KUKA KRL program: MyProgram_213().src

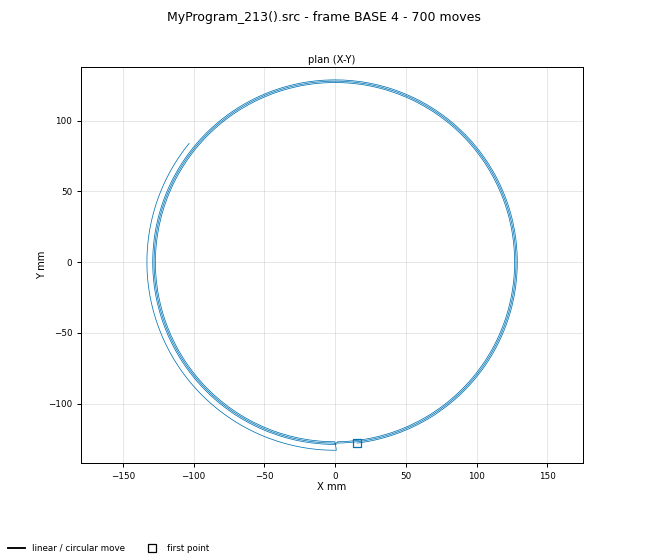
[picture p0: tool path of MyProgram_213().src in frame BASE 4, 700 of 700 moves have a stored position in this frame; points joined in program order, loops and branches not executed]
&ACCESS RVP
&REL 1
&PARAM TEMPLATE = C:\KRC\Roboter\Template\vorgabe
&PARAM EDITMASK = *
DEF MyProgram_213()
; ---- Setting reference (Base) ----
$BASE = BASE_DATA[4]

; --------------------------
; ---- Setting tool (TCP) ----
$TOOL = TOOL_DATA[3]
; --------------------------

$VEL.CP = VEL_APROX_PRINT
Startdeposition()
$VEL.CP = VEL_PRINT
LIN {X 15.6631,Y -127.8764,Z 150,A -84.7051,B 21.2641,C -0.7422,E1 21.2973,E2 532.2329} C_DIS
LIN {X 18.2596,Y -127.5309,Z 150,A -82.9319,B 21.2632,C -0.7696,E1 21.3024,E2 530.386} C_DIS
LIN {X 22.8874,Y -126.7822,Z 150,A -81.4703,B 21.2641,C -0.7437,E1 21.3063,E2 528.9976} C_DIS
LIN {X 26.4582,Y -126.0874,Z 150,A -79.8315,B 21.2641,C -0.746,E1 21.3107,E2 527.3551} C_DIS
LIN {X 29.8823,Y -125.3182,Z 150,A -78.1484,B 21.2638,C -0.7528,E1 21.3154,E2 525.6559} C_DIS
LIN {X 34.3471,Y -124.1689,Z 150,A -76.3006,B 21.264,C -0.746,E1 21.3203,E2 523.8305} C_DIS
LIN {X 37.1802,Y -123.3508,Z 150,A -74.8395,B 21.2637,C -0.754,E1 21.3243,E2 522.3503} C_DIS
LIN {X 39.8601,Y -122.5118,Z 150,A -73.2468,B 21.2632,C -0.7707,E1 21.3286,E2 520.7152} C_DIS
LIN {X 43.4,Y -121.3013,Z 150,A -71.878,B 21.2635,C -0.7597,E1 21.3321,E2 519.3802} C_DIS
LIN {X 46.1763,Y -120.2726,Z 150,A -69.6143,B 21.262,C -0.8039,E1 21.3384,E2 517.0006} C_DIS
LIN {X 52.7771,Y -117.5247,Z 150,A -67.5502,B 21.2636,C -0.7583,E1 21.3433,E2 515.068} C_DIS
LIN {X 56.4516,Y -115.806,Z 150,A -65.6853,B 21.2634,C -0.7638,E1 21.348,E2 513.1938} C_DIS
LIN {X 59.7288,Y -114.1488,Z 150,A -64.1905,B 21.2635,C -0.7603,E1 21.3516,E2 511.7136} C_DIS
LIN {X 62.0762,Y -112.8921,Z 150,A -62.4263,B 21.2625,C -0.7884,E1 21.3561,E2 509.8784} C_DIS
LIN {X 65.7163,Y -110.8119,Z 150,A -60.7738,B 21.2628,C -0.7822,E1 21.3601,E2 508.2491} C_DIS
LIN {X 68.4873,Y -109.1217,Z 150,A -59.507,B 21.2629,C -0.7768,E1 21.363,E2 507.0018} C_DIS
LIN {X 72.1434,Y -106.7393,Z 150,A -57.4433,B 21.2626,C -0.7862,E1 21.3678,E2 504.9208} C_DIS
LIN {X 79.2097,Y -101.6066,Z 150,A -52.9654,B 21.2614,C -0.8213,E1 21.378,E2 500.3657} C_DIS
LIN {X 83.9285,Y -97.7445,Z 150,A -51.3313,B 21.2629,C -0.7781,E1 21.3812,E2 498.8579} C_DIS
LIN {X 88.2018,Y -93.9067,Z 150,A -48.6114,B 21.2624,C -0.7913,E1 21.3869,E2 496.1147} C_DIS
LIN {X 93.8183,Y -88.2955,Z 150,A -45.2617,B 21.2624,C -0.7915,E1 21.3935,E2 492.7815} C_DIS
LIN {X 97.7896,Y -83.8762,Z 150,A -42.3753,B 21.2618,C -0.8092,E1 21.3989,E2 489.8621} C_DIS
LIN {X 100.2723,Y -80.8914,Z 150,A -39.8306,B 21.2602,C -0.8514,E1 21.4035,E2 487.2158} C_DIS
LIN {X 104.1395,Y -75.8485,Z 150,A -37.8772,B 21.2615,C -0.8186,E1 21.4066,E2 485.3636} C_DIS
LIN {X 106.3473,Y -72.7204,Z 150,A -36.1507,B 21.2612,C -0.8244,E1 21.4093,E2 483.6315} C_DIS
LIN {X 108.4584,Y -69.5322,Z 150,A -34.4696,B 21.2612,C -0.8282,E1 21.4119,E2 481.95} C_DIS
LIN {X 110.584,Y -66.0994,Z 150,A -32.5234,B 21.2607,C -0.8402,E1 21.4147,E2 479.9828} C_DIS
LIN {X 113.2426,Y -61.434,Z 150,A -30.2698,B 21.2607,C -0.8408,E1 21.4178,E2 477.7415} C_DIS
LIN {X 114.9781,Y -58.1173,Z 150,A -28.251,B 21.2598,C -0.8621,E1 21.4204,E2 475.6772} C_DIS
LIN {X 116.8181,Y -54.3235,Z 150,A -26.8866,B 21.2605,C -0.844,E1 21.4219,E2 474.3712} C_DIS
LIN {X 118.3125,Y -50.9865,Z 150,A -25.2141,B 21.2602,C -0.851,E1 21.4238,E2 472.6904} C_DIS
LIN {X 119.5881,Y -47.9188,Z 150,A -23.3605,B 21.2594,C -0.8729,E1 21.4258,E2 470.7892} C_DIS
LIN {X 121.0232,Y -44.1714,Z 150,A -21.9784,B 21.2599,C -0.8597,E1 21.4271,E2 469.4525} C_DIS
LIN {X 122.1969,Y -40.8095,Z 150,A -20.5058,B 21.2599,C -0.8594,E1 21.4284,E2 467.9905} C_DIS
LIN {X 123.1384,Y -37.8741,Z 150,A -18.6791,B 21.2589,C -0.8848,E1 21.4299,E2 466.1068} C_DIS
LIN {X 124.2425,Y -34.084,Z 150,A -17.3486,B 21.2595,C -0.8705,E1 21.4309,E2 464.8245} C_DIS
LIN {X 125.1127,Y -30.7349,Z 150,A -15.7365,B 21.2592,C -0.8787,E1 21.432,E2 463.2011} C_DIS
LIN {X 125.9433,Y -27.1259,Z 150,A -14.1941,B 21.2592,C -0.8791,E1 21.4329,E2 461.6684} C_DIS
LIN {X 126.4726,Y -24.5423,Z 150,A -12.9669,B 21.2589,C -0.8853,E1 21.4336,E2 460.4328} C_DIS
LIN {X 127.608,Y -17.7203,Z 150,A -10.3865,B 21.2594,C -0.8721,E1 21.4348,E2 457.9065} C_DIS
LIN {X 128.361,Y -11.0017,Z 150,A -7.2717,B 21.2589,C -0.8865,E1 21.4357,E2 454.7743} C_DIS
LIN {X 128.759,Y -4.3743,Z 150,A -4.1384,B 21.2581,C -0.9042,E1 21.4362,E2 451.615} C_DIS
LIN {X 128.8171,Y 1.9443,Z 150,A -0.5419,B 21.2563,C -0.9496,E1 21.4362,E2 447.9196} C_DIS
LIN {X 128.6186,Y 7.4224,Z 150,A 1.2036,B 21.2573,C -0.9251,E1 21.4359,E2 446.2535} C_DIS
LIN {X 127.9217,Y 15.2834,Z 150,A 4.5209,B 21.2572,C -0.9273,E1 21.4351,E2 442.9539} C_DIS
LIN {X 127.0644,Y 21.2642,Z 150,A 7.3154,B 21.2566,C -0.9405,E1 21.4339,E2 440.1427} C_DIS
LIN {X 125.7034,Y 28.2204,Z 150,A 10.2724,B 21.2566,C -0.9412,E1 21.4323,E2 437.2044} C_DIS
LIN {X 125.0364,Y 31.0459,Z 150,A 11.7612,B 21.2561,C -0.9542,E1 21.4313,E2 435.6903} C_DIS
LIN {X 124.0877,Y 34.6374,Z 150,A 13.3155,B 21.2561,C -0.9548,E1 21.4301,E2 434.1453} C_DIS
LIN {X 123.0525,Y 38.1549,Z 150,A 15.0849,B 21.2556,C -0.966,E1 21.4287,E2 432.3572} C_DIS
LIN {X 121.7679,Y 42.0723,Z 150,A 16.7524,B 21.2556,C -0.9638,E1 21.4272,E2 430.7069} C_DIS
LIN {X 120.5533,Y 45.4363,Z 150,A 18.342,B 21.2554,C -0.9684,E1 21.4257,E2 429.1154} C_DIS
LIN {X 118.9128,Y 49.5703,Z 150,A 20.4851,B 21.2549,C -0.9817,E1 21.4234,E2 426.9501} C_DIS
LIN {X 116.9548,Y 54.0279,Z 150,A 22.3283,B 21.2552,C -0.9731,E1 21.4213,E2 425.1424} C_DIS
LIN {X 115.3134,Y 57.4502,Z 150,A 24.2806,B 21.2545,C -0.9898,E1 21.4189,E2 423.1567} C_DIS
LIN {X 113.262,Y 61.3985,Z 150,A 26.1914,B 21.2545,C -0.9921,E1 21.4164,E2 421.2517} C_DIS
LIN {X 111.2644,Y 64.9485,Z 150,A 28.5674,B 21.253,C -1.0227,E1 21.413,E2 418.8065} C_DIS
LIN {X 108.6614,Y 69.2151,Z 150,A 30.0028,B 21.2544,C -0.9926,E1 21.411,E2 417.4623} C_DIS
LIN {X 105.2657,Y 74.277,Z 150,A 32.9043,B 21.2537,C -1.008,E1 21.4064,E2 414.5356} C_DIS
LIN {X 102.595,Y 77.9254,Z 150,A 34.8935,B 21.2535,C -1.012,E1 21.4031,E2 412.547} C_DIS
LIN {X 100.0939,Y 81.1125,Z 150,A 36.7233,B 21.2533,C -1.0175,E1 21.3999,E2 410.7122} C_DIS
LIN {X 97.298,Y 84.4462,Z 150,A 38.6614,B 21.253,C -1.0221,E1 21.3964,E2 408.772} C_DIS
LIN {X 94.2248,Y 87.8615,Z 150,A 41.093,B 21.252,C -1.0442,E1 21.3917,E2 406.2927} C_DIS
LIN {X 91.1719,Y 91.0259,Z 150,A 42.3252,B 21.2533,C -1.0159,E1 21.3894,E2 405.1445} C_DIS
LIN {X 86.1606,Y 95.7829,Z 150,A 45.6877,B 21.2525,C -1.0351,E1 21.3825,E2 401.7458} C_DIS
LIN {X 82.649,Y 98.8288,Z 150,A 47.7085,B 21.2524,C -1.037,E1 21.3782,E2 399.7292} C_DIS
LIN {X 79.3182,Y 101.5218,Z 150,A 49.6298,B 21.2522,C -1.0412,E1 21.374,E2 397.8048} C_DIS
LIN {X 75.866,Y 104.1268,Z 150,A 51.5463,B 21.252,C -1.0443,E1 21.3697,E2 395.888} C_DIS
LIN {X 71.0796,Y 107.451,Z 150,A 54.1358,B 21.2518,C -1.0485,E1 21.3637,E2 393.2976} C_DIS
LIN {X 66.8868,Y 110.1098,Z 150,A 56.5776,B 21.2512,C -1.0622,E1 21.3578,E2 390.8273} C_DIS
LIN {X 63.8693,Y 111.8868,Z 150,A 57.8348,B 21.2517,C -1.0512,E1 21.3549,E2 389.6048} C_DIS
LIN {X 60.1767,Y 113.9136,Z 150,A 59.5718,B 21.2519,C -1.0478,E1 21.3506,E2 387.8831} C_DIS
LIN {X 55.6959,Y 116.1699,Z 150,A 61.8479,B 21.2516,C -1.0526,E1 21.3449,E2 385.6012} C_DIS
LIN {X 52.6861,Y 117.5654,Z 150,A 63.1504,B 21.2519,C -1.0468,E1 21.3417,E2 384.3187} C_DIS
LIN {X 50.3275,Y 118.5962,Z 150,A 64.7065,B 21.251,C -1.066,E1 21.3376,E2 382.7143} C_DIS
LIN {X 47.1871,Y 119.8797,Z 150,A 66.2089,B 21.251,C -1.0672,E1 21.3337,E2 381.2125} C_DIS
LIN {X 42.4741,Y 121.6286,Z 150,A 68.2256,B 21.2513,C -1.0598,E1 21.3284,E2 379.2212} C_DIS
LIN {X 39.205,Y 122.721,Z 150,A 69.7604,B 21.2513,C -1.0611,E1 21.3244,E2 377.6861} C_DIS
LIN {X 35.6855,Y 123.7915,Z 150,A 71.4929,B 21.251,C -1.0665,E1 21.3197,E2 375.9424} C_DIS
LIN {X 31.8313,Y 124.8371,Z 150,A 73.1584,B 21.2511,C -1.0629,E1 21.3152,E2 374.2899} C_DIS
LIN {X 28.5909,Y 125.6188,Z 150,A 74.8391,B 21.2507,C -1.0723,E1 21.3106,E2 372.5863} C_DIS
LIN {X 23.7855,Y 126.6173,Z 150,A 76.9127,B 21.2509,C -1.0686,E1 21.3049,E2 370.5258} C_DIS
LIN {X 18.8801,Y 127.4422,Z 150,A 79.1764,B 21.2507,C -1.0715,E1 21.2987,E2 368.2567} C_DIS
LIN {X 11.8911,Y 128.2823,Z 150,A 82.2359,B 21.2508,C -1.0691,E1 21.2902,E2 365.2065} C_DIS
LIN {X 5.5858,Y 128.7117,Z 150,A 84.8426,B 21.2513,C -1.0605,E1 21.283,E2 362.6248} C_DIS
LIN {X -0.8667,Y 128.8288,Z 150,A 87.7032,B 21.2513,C -1.0597,E1 21.2751,E2 359.7667} C_DIS
LIN {X -7.8241,Y 128.5938,Z 150,A 90.6265,B 21.2517,C -1.0516,E1 21.267,E2 356.8653} C_DIS
LIN {X -14.0882,Y 128.0593,Z 150,A 93.8551,B 21.2509,C -1.0683,E1 21.2579,E2 353.5886} C_DIS
LIN {X -19.8208,Y 127.2976,Z 150,A 96.6448,B 21.2505,C -1.0758,E1 21.2501,E2 350.7754} C_DIS
LIN {X -23.2891,Y 126.7103,Z 150,A 98.0736,B 21.2508,C -1.069,E1 21.2462,E2 349.3637} C_DIS
LIN {X -27.6706,Y 125.8257,Z 150,A 99.8943,B 21.2513,C -1.0605,E1 21.2413,E2 347.564} C_DIS
LIN {X -31.5061,Y 124.9196,Z 150,A 101.6318,B 21.2513,C -1.0583,E1 21.2366,E2 345.8296} C_DIS
LIN {X -35.0763,Y 123.9649,Z 150,A 103.3914,B 21.2513,C -1.0614,E1 21.2318,E2 344.0582} C_DIS
LIN {X -39.4365,Y 122.6471,Z 150,A 105.9866,B 21.2502,C -1.0827,E1 21.2247,E2 341.3985} C_DIS
LIN {X -44.4011,Y 120.9404,Z 150,A 107.7786,B 21.2514,C -1.0574,E1 21.2202,E2 339.6723} C_DIS
LIN {X -48.0505,Y 119.5351,Z 150,A 109.4231,B 21.2517,C -1.0513,E1 21.2159,E2 338.0404} C_DIS
LIN {X -51.2634,Y 118.1928,Z 150,A 110.8864,B 21.252,C -1.0456,E1 21.2122,E2 336.5887} C_DIS
LIN {X -53.5532,Y 117.1744,Z 150,A 112.2903,B 21.2515,C -1.0558,E1 21.2086,E2 335.1525} C_DIS
LIN {X -58.166,Y 114.9533,Z 150,A 114.3393,B 21.2521,C -1.043,E1 21.2035,E2 333.1325} C_DIS
LIN {X -63.2468,Y 112.24,Z 150,A 116.9999,B 21.2521,C -1.0427,E1 21.197,E2 330.4637} C_DIS
LIN {X -66.0415,Y 110.6186,Z 150,A 118.7425,B 21.2516,C -1.0526,E1 21.1927,E2 328.6874} C_DIS
LIN {X -69.1561,Y 108.6992,Z 150,A 120.1279,B 21.2522,C -1.0398,E1 21.1895,E2 327.3321} C_DIS
LIN {X -72.9552,Y 106.1861,Z 150,A 121.9941,B 21.2527,C -1.0295,E1 21.1852,E2 325.4869} C_DIS
LIN {X -75.6796,Y 104.2619,Z 150,A 123.5721,B 21.2527,C -1.0304,E1 21.1816,E2 323.9} C_DIS
LIN {X -80.5249,Y 100.5675,Z 150,A 126.3636,B 21.2527,C -1.028,E1 21.1755,E2 321.1028} C_DIS
LIN {X -83.5461,Y 98.0715,Z 150,A 128.2062,B 21.2527,C -1.0282,E1 21.1715,E2 319.2511} C_DIS
LIN {X -87.9544,Y 94.1382,Z 150,A 130.7275,B 21.2532,C -1.018,E1 21.1663,E2 316.7459} C_DIS
LIN {X -91.0627,Y 91.1354,Z 150,A 132.6952,B 21.2534,C -1.0154,E1 21.1624,E2 314.7758} C_DIS
LIN {X -95.0812,Y 86.9346,Z 150,A 135.1717,B 21.2538,C -1.0048,E1 21.1577,E2 312.3157} C_DIS
LIN {X -97.7706,Y 83.8982,Z 150,A 137.0559,B 21.2538,C -1.0034,E1 21.1542,E2 310.425} C_DIS
LIN {X -100.4242,Y 80.703,Z 150,A 139.0535,B 21.2538,C -1.0047,E1 21.1507,E2 308.4129} C_DIS
LIN {X -103.0555,Y 77.3151,Z 150,A 140.7212,B 21.2545,C -0.9902,E1 21.1479,E2 306.7759} C_DIS
LIN {X -106.0447,Y 73.1612,Z 150,A 143.0774,B 21.2546,C -0.9872,E1 21.1441,E2 304.4141} C_DIS
LIN {X -108.3199,Y 69.7483,Z 150,A 144.9588,B 21.2547,C -0.9844,E1 21.1412,E2 302.529} C_DIS
LIN {X -109.8587,Y 67.2981,Z 150,A 147.162,B 21.2533,C -1.0172,E1 21.1379,E2 300.2212} C_DIS
LIN {X -113.1387,Y 61.6247,Z 150,A 148.9226,B 21.2557,C -0.9632,E1 21.1357,E2 298.5995} C_DIS
LIN {X -114.9418,Y 58.1885,Z 150,A 151.795,B 21.2539,C -1.0035,E1 21.1319,E2 295.5968} C_DIS
LIN {X -117.6656,Y 52.4623,Z 150,A 153.6951,B 21.2559,C -0.9587,E1 21.1298,E2 293.8085} C_DIS
LIN {X -119.153,Y 48.9951,Z 150,A 155.5188,B 21.2559,C -0.9594,E1 21.1278,E2 291.9708} C_DIS
LIN {X -120.4519,Y 45.7069,Z 150,A 156.9715,B 21.2562,C -0.95,E1 21.1264,E2 290.5346} C_DIS
LIN {X -121.8856,Y 41.7327,Z 150,A 158.9914,B 21.2562,C -0.9498,E1 21.1245,E2 288.5015} C_DIS
LIN {X -123.9974,Y 34.9595,Z 150,A 162.1389,B 21.2567,C -0.9397,E1 21.122,E2 285.3602} C_DIS
LIN {X -125.1447,Y 30.6021,Z 150,A 164.1,B 21.257,C -0.9318,E1 21.1206,E2 283.4074} C_DIS
LIN {X -125.877,Y 27.4328,Z 150,A 165.3473,B 21.2575,C -0.9195,E1 21.1198,E2 282.1855} C_DIS
LIN {X -126.5003,Y 24.3974,Z 150,A 166.9854,B 21.2573,C -0.9253,E1 21.1189,E2 280.5196} C_DIS
LIN {X -127.2132,Y 20.3664,Z 150,A 168.8409,B 21.2575,C -0.9209,E1 21.1181,E2 278.6631} C_DIS
LIN {X -127.7347,Y 16.7746,Z 150,A 170.3092,B 21.2579,C -0.9101,E1 21.1175,E2 277.2143} C_DIS
LIN {X -128.1819,Y 12.9363,Z 150,A 172.1716,B 21.2579,C -0.9102,E1 21.117,E2 275.3382} C_DIS
LIN {X -128.5728,Y 8.1646,Z 150,A 174.2415,B 21.2583,C -0.9011,E1 21.1165,E2 273.2786} C_DIS
LIN {X -128.7429,Y 4.7847,Z 150,A 175.6056,B 21.2587,C -0.8908,E1 21.1164,E2 271.9332} C_DIS
LIN {X -128.8283,Y 1.0282,Z 150,A 177.769,B 21.2581,C -0.9048,E1 21.1163,E2 269.7153} C_DIS
LIN {X -128.7807,Y -3.6216,Z 150,A 179.5823,B 21.2588,C -0.8882,E1 21.1163,E2 267.935} C_DIS
LIN {X -128.5928,Y -7.8404,Z 150,A -178.5359,B 21.259,C -0.8825,E1 21.1166,E2 266.0557} C_DIS
LIN {X -128.3283,Y -11.3896,Z 150,A -177.1068,B 21.2595,C -0.8714,E1 21.117,E2 264.6468} C_DIS
LIN {X -127.8524,Y -15.8644,Z 150,A -174.8329,B 21.2593,C -0.8758,E1 21.1177,E2 262.3444} C_DIS
LIN {X -127.3145,Y -19.7116,Z 150,A -173.2072,B 21.2596,C -0.8665,E1 21.1183,E2 260.7332} C_DIS
LIN {X -126.6665,Y -23.528,Z 150,A -171.3296,B 21.2596,C -0.8673,E1 21.1193,E2 258.84} C_DIS
LIN {X -125.8908,Y -27.3689,Z 150,A -169.6939,B 21.26,C -0.8577,E1 21.1202,E2 257.2192} C_DIS
LIN {X -124.9367,Y -31.4386,Z 150,A -167.9395,B 21.2604,C -0.8479,E1 21.1213,E2 255.4797} C_DIS
LIN {X -124.0968,Y -34.6048,Z 150,A -166.4306,B 21.2604,C -0.8456,E1 21.1224,E2 253.9667} C_DIS
LIN {X -123.2133,Y -37.6295,Z 150,A -164.9638,B 21.2605,C -0.844,E1 21.1236,E2 252.4942} C_DIS
LIN {X -121.594,Y -42.573,Z 150,A -162.3671,B 21.2603,C -0.8484,E1 21.126,E2 249.8676} C_DIS
LIN {X -120.3324,Y -46.0227,Z 150,A -160.6938,B 21.2605,C -0.8452,E1 21.1277,E2 248.1919} C_DIS
LIN {X -118.3246,Y -50.9586,Z 150,A -158.597,B 21.2611,C -0.8276,E1 21.1299,E2 246.13} C_DIS
LIN {X -117.0785,Y -53.7606,Z 150,A -157.2037,B 21.2612,C -0.8249,E1 21.1315,E2 244.7351} C_DIS
LIN {X -115.5673,Y -56.9355,Z 150,A -155.671,B 21.2614,C -0.8193,E1 21.1333,E2 243.2078} C_DIS
LIN {X -113.9962,Y -60.0193,Z 150,A -153.7044,B 21.261,C -0.8322,E1 21.1359,E2 241.193} C_DIS
LIN {X -112.153,Y -63.4016,Z 150,A -152.2664,B 21.2615,C -0.8166,E1 21.1379,E2 239.7893} C_DIS
LIN {X -109.829,Y -67.3464,Z 150,A -150.2799,B 21.2618,C -0.8092,E1 21.1407,E2 237.8109} C_DIS
LIN {X -107.5121,Y -70.9868,Z 150,A -148.3723,B 21.262,C -0.8038,E1 21.1436,E2 235.9067} C_DIS
LIN {X -105.163,Y -74.4226,Z 150,A -146.4491,B 21.262,C -0.8021,E1 21.1467,E2 233.9769} C_DIS
LIN {X -102.6277,Y -77.8821,Z 150,A -144.5434,B 21.2622,C -0.7974,E1 21.1498,E2 232.0733} C_DIS
LIN {X -100.0395,Y -81.18,Z 150,A -142.6257,B 21.2623,C -0.7951,E1 21.1532,E2 230.1511} C_DIS
LIN {X -97.2154,Y -84.5409,Z 150,A -140.8196,B 21.2627,C -0.7848,E1 21.1564,E2 228.3639} C_DIS
LIN {X -93.8865,Y -88.2232,Z 150,A -138.4741,B 21.2627,C -0.7855,E1 21.1609,E2 226.0041} C_DIS
LIN {X -90.9577,Y -91.2397,Z 150,A -136.5766,B 21.2627,C -0.7826,E1 21.1646,E2 224.1049} C_DIS
LIN {X -87.7302,Y -94.347,Z 150,A -134.6214,B 21.2629,C -0.777,E1 21.1686,E2 222.1555} C_DIS
LIN {X -84.5261,Y -97.2283,Z 150,A -132.6674,B 21.263,C -0.7748,E1 21.1727,E2 220.1984} C_DIS
LIN {X -81.281,Y -99.9572,Z 150,A -130.7547,B 21.2631,C -0.7724,E1 21.1768,E2 218.2837} C_DIS
LIN {X -77.8909,Y -102.621,Z 150,A -128.5206,B 21.2628,C -0.782,E1 21.1818,E2 216.0133} C_DIS
LIN {X -74.8985,Y -104.8244,Z 150,A -127.1603,B 21.2633,C -0.7671,E1 21.1848,E2 214.6884} C_DIS
LIN {X -71.0904,Y -107.4439,Z 150,A -125.089,B 21.2633,C -0.7645,E1 21.1896,E2 212.6162} C_DIS
LIN {X -68.4461,Y -109.1477,Z 150,A -123.675,B 21.2634,C -0.7629,E1 21.193,E2 211.201} C_DIS
LIN {X -64.6494,Y -111.4379,Z 150,A -121.7472,B 21.2636,C -0.7583,E1 21.1976,E2 209.2792} C_DIS
LIN {X -60.9578,Y -113.4993,Z 150,A -119.7837,B 21.2636,C -0.7592,E1 21.2024,E2 207.3065} C_DIS
LIN {X -57.0758,Y -115.4981,Z 150,A -118.121,B 21.264,C -0.7452,E1 21.2065,E2 205.6773} C_DIS
LIN {X -53.565,Y -117.1689,Z 150,A -115.9371,B 21.2635,C -0.7621,E1 21.2121,E2 203.44} C_DIS
LIN {X -50.5191,Y -118.5146,Z 150,A -114.4503,B 21.2635,C -0.7608,E1 21.216,E2 201.9527} C_DIS
LIN {X -47.4144,Y -119.7913,Z 150,A -113.1335,B 21.2638,C -0.7519,E1 21.2193,E2 200.657} C_DIS
LIN {X -43.7757,Y -121.1659,Z 150,A -111.5396,B 21.264,C -0.7446,E1 21.2235,E2 199.0793} C_DIS
LIN {X -40.9362,Y -122.1547,Z 150,A -110.3003,B 21.2642,C -0.7394,E1 21.2267,E2 197.8517} C_DIS
LIN {X -37.8224,Y -123.1542,Z 150,A -108.7565,B 21.2642,C -0.7421,E1 21.2308,E2 196.2973} C_DIS
LIN {X -35.2104,Y -123.9274,Z 150,A -107.5103,B 21.2642,C -0.7427,E1 21.2342,E2 195.047} C_DIS
LIN {X -31.803,Y -124.8442,Z 150,A -106.2025,B 21.2645,C -0.7307,E1 21.2376,E2 193.77} C_DIS
LIN {X -28.1024,Y -125.7304,Z 150,A -104.1717,B 21.2641,C -0.7441,E1 21.2433,E2 191.699} C_DIS
LIN {X -24.3505,Y -126.5093,Z 150,A -102.5584,B 21.2642,C -0.7395,E1 21.2477,E2 190.0961} C_DIS
LIN {X -21.2575,Y -127.0656,Z 150,A -101.2585,B 21.2644,C -0.7349,E1 21.2512,E2 188.8075} C_DIS
LIN {X -17.0537,Y -127.6982,Z 150,A -99.1457,B 21.2641,C -0.7439,E1 21.2571,E2 186.6678} C_DIS
LIN {X -9.2958,Y -128.4958,Z 150,A -95.9473,B 21.2645,C -0.7319,E1 21.2659,E2 183.5005} C_DIS
LIN {X -4.3113,Y -128.7614,Z 150,A -93.4511,B 21.2641,C -0.7439,E1 21.273,E2 180.9705} C_DIS
LIN {X 0.9222,Y -128.7994,Z 150,A -91.6037,B 21.2647,C -0.724,E1 21.278,E2 179.1779} C_DIS
Enddeposition()
LIN {X 0.9222,Y -128.7994,Z 150,A -91.6037,B 21.2647,C -0.724,E1 21.278,E2 179.1779} C_DIS
Startdeposition()
$VEL.CP = VEL_PRINT
LIN {X -0.4498,Y -127.8841,Z 150,A -92.2338,B 20.0862,C -0.5518,E1 20.0922,E2 180.1706} C_DIS
LIN {X -6.976,Y -127.6954,Z 150,A -95.1395,B 20.0862,C -0.5523,E1 20.084,E2 183.0755} C_DIS
LIN {X -10.8958,Y -127.4196,Z 150,A -96.8501,B 20.0861,C -0.5544,E1 20.0793,E2 184.7809} C_DIS
LIN {X -14.5522,Y -127.0553,Z 150,A -98.8648,B 20.0865,C -0.5401,E1 20.0736,E2 186.8388} C_DIS
LIN {X -17.8229,Y -126.6367,Z 150,A -100.1255,B 20.0862,C -0.549,E1 20.0702,E2 188.0749} C_DIS
LIN {X -22.5021,Y -125.8892,Z 150,A -102.1325,B 20.0862,C -0.5542,E1 20.0647,E2 190.069} C_DIS
LIN {X -25.7127,Y -125.273,Z 150,A -103.6706,B 20.0862,C -0.552,E1 20.0604,E2 191.6159} C_DIS
LIN {X -30.1019,Y -124.2912,Z 150,A -105.5988,B 20.086,C -0.5564,E1 20.0552,E2 193.5343} C_DIS
LIN {X -33.6569,Y -123.378,Z 150,A -107.4107,B 20.0862,C -0.5509,E1 20.0503,E2 195.3658} C_DIS
LIN {X -37.7481,Y -122.1867,Z 150,A -109.2912,B 20.0862,C -0.5534,E1 20.0452,E2 197.243} C_DIS
LIN {X -41.7643,Y -120.8724,Z 150,A -111.0605,B 20.086,C -0.5598,E1 20.0406,E2 198.9979} C_DIS
LIN {X -44.8587,Y -119.7583,Z 150,A -112.5326,B 20.086,C -0.5611,E1 20.0367,E2 200.4699} C_DIS
LIN {X -48.1557,Y -118.4716,Z 150,A -114.2228,B 20.086,C -0.5587,E1 20.0323,E2 202.1719} C_DIS
LIN {X -52.3698,Y -116.6695,Z 150,A -116.1907,B 20.0858,C -0.5642,E1 20.0273,E2 204.1297} C_DIS
LIN {X -55.8021,Y -115.0697,Z 150,A -117.8743,B 20.0858,C -0.5666,E1 20.0231,E2 205.8115} C_DIS
LIN {X -58.2849,Y -113.8301,Z 150,A -119.1593,B 20.0858,C -0.5666,E1 20.0198,E2 207.101} C_DIS
LIN {X -61.7243,Y -112.0046,Z 150,A -120.9399,B 20.0858,C -0.5675,E1 20.0155,E2 208.8853} C_DIS
LIN {X -65.2299,Y -109.9999,Z 150,A -122.832,B 20.0858,C -0.567,E1 20.0109,E2 210.7863} C_DIS
LIN {X -68.9933,Y -107.679,Z 150,A -124.685,B 20.0855,C -0.5748,E1 20.0065,E2 212.6238} C_DIS
LIN {X -72.1049,Y -105.6211,Z 150,A -126.5031,B 20.0856,C -0.5719,E1 20.0023,E2 214.4581} C_DIS
LIN {X -75.6823,Y -103.0875,Z 150,A -128.4771,B 20.0856,C -0.5749,E1 19.9978,E2 216.4322} C_DIS
LIN {X -78.2281,Y -101.1692,Z 150,A -129.8892,B 20.0855,C -0.578,E1 19.9947,E2 217.8418} C_DIS
LIN {X -81.7344,Y -98.3584,Z 150,A -131.869,B 20.0853,C -0.5829,E1 19.9904,E2 219.8166} C_DIS
LIN {X -84.7576,Y -95.7652,Z 150,A -133.6886,B 20.0853,C -0.585,E1 19.9866,E2 221.639} C_DIS
LIN {X -87.952,Y -92.8404,Z 150,A -135.6618,B 20.0852,C -0.5877,E1 19.9825,E2 223.6147} C_DIS
LIN {X -90.8841,Y -89.972,Z 150,A -137.5009,B 20.0851,C -0.5915,E1 19.9789,E2 225.4526} C_DIS
LIN {X -93.6278,Y -87.113,Z 150,A -139.2718,B 20.085,C -0.5955,E1 19.9755,E2 227.2217} C_DIS
LIN {X -95.9851,Y -84.5089,Z 150,A -140.8525,B 20.0849,C -0.5987,E1 19.9726,E2 228.8019} C_DIS
LIN {X -98.693,Y -81.3302,Z 150,A -142.753,B 20.0848,C -0.6019,E1 19.9692,E2 230.7042} C_DIS
LIN {X -101.3994,Y -77.93,Z 150,A -144.7378,B 20.0847,C -0.6051,E1 19.9657,E2 232.6916} C_DIS
LIN {X -103.8313,Y -74.6594,Z 150,A -146.5727,B 20.0846,C -0.6092,E1 19.9627,E2 234.5258} C_DIS
LIN {X -106.3397,Y -71.0401,Z 150,A -148.5095,B 20.0844,C -0.6155,E1 19.9597,E2 236.4565} C_DIS
LIN {X -108.2732,Y -68.0574,Z 150,A -150.1286,B 20.0844,C -0.6186,E1 19.9573,E2 238.077} C_DIS
LIN {X -110.2616,Y -64.786,Z 150,A -151.8442,B 20.0842,C -0.623,E1 19.9548,E2 239.7909} C_DIS
LIN {X -112.3363,Y -61.1181,Z 150,A -153.8048,B 20.0841,C -0.6254,E1 19.9521,E2 241.7577} C_DIS
LIN {X -114.084,Y -57.7861,Z 150,A -155.3356,B 20.0838,C -0.6356,E1 19.9502,E2 243.2689} C_DIS
LIN {X -115.4947,Y -54.9124,Z 150,A -156.7941,B 20.0837,C -0.6387,E1 19.9484,E2 244.7286} C_DIS
LIN {X -117.028,Y -51.5684,Z 150,A -158.4407,B 20.0836,C -0.6433,E1 19.9465,E2 246.3731} C_DIS
LIN {X -118.2507,Y -48.6983,Z 150,A -159.9891,B 20.0836,C -0.6418,E1 19.9449,E2 247.937} C_DIS
LIN {X -119.4267,Y -45.7387,Z 150,A -161.2547,B 20.0833,C -0.6517,E1 19.9436,E2 249.1825} C_DIS
LIN {X -121.4588,Y -40.0286,Z 150,A -164.0473,B 20.0831,C -0.6568,E1 19.941,E2 251.9805} C_DIS
LIN {X -122.7327,Y -35.9313,Z 150,A -166.0353,B 20.0831,C -0.6601,E1 19.9394,E2 253.9734} C_DIS
LIN {X -123.7065,Y -32.4253,Z 150,A -167.5898,B 20.0828,C -0.6677,E1 19.9383,E2 255.5172} C_DIS
LIN {X -124.5954,Y -28.8185,Z 150,A -169.3066,B 20.0827,C -0.6708,E1 19.9371,E2 257.2377} C_DIS
LIN {X -125.3041,Y -25.5598,Z 150,A -170.8161,B 20.0826,C -0.6748,E1 19.9363,E2 258.7468} C_DIS
LIN {X -126.0127,Y -21.8116,Z 150,A -172.6664,B 20.0826,C -0.6749,E1 19.9354,E2 260.6108} C_DIS
LIN {X -126.6118,Y -17.9972,Z 150,A -174.3054,B 20.0823,C -0.6835,E1 19.9347,E2 262.2369} C_DIS
LIN {X -127.1423,Y -13.7585,Z 150,A -176.149,B 20.082,C -0.692,E1 19.9341,E2 264.0698} C_DIS
LIN {X -127.4569,Y -10.4541,Z 150,A -177.6841,B 20.082,C -0.6949,E1 19.9337,E2 265.6082} C_DIS
LIN {X -127.7141,Y -6.6038,Z 150,A -179.5251,B 20.0819,C -0.6962,E1 19.9334,E2 267.4594} C_DIS
LIN {X -127.8577,Y -2.6856,Z 150,A 178.6219,B 20.0818,C -0.6983,E1 19.9332,E2 269.3206} C_DIS
LIN {X -127.868,Y 2.0641,Z 150,A 176.6805,B 20.0813,C -0.7117,E1 19.9332,E2 271.2377} C_DIS
LIN {X -127.7588,Y 5.7157,Z 150,A 175.0217,B 20.0812,C -0.716,E1 19.9334,E2 272.8965} C_DIS
LIN {X -127.6031,Y 8.5045,Z 150,A 173.5469,B 20.0813,C -0.7119,E1 19.9337,E2 274.3946} C_DIS
LIN {X -127.2894,Y 12.3242,Z 150,A 171.9031,B 20.0811,C -0.72,E1 19.9341,E2 276.0274} C_DIS
LIN {X -126.7837,Y 16.7438,Z 150,A 169.9597,B 20.0808,C -0.728,E1 19.9348,E2 277.9621} C_DIS
LIN {X -126.3445,Y 19.7876,Z 150,A 168.6066,B 20.0806,C -0.7332,E1 19.9353,E2 279.3103} C_DIS
LIN {X -125.6783,Y 23.6542,Z 150,A 166.7518,B 20.0806,C -0.7352,E1 19.9362,E2 281.1732} C_DIS
LIN {X -125.0055,Y 26.9821,Z 150,A 165.24,B 20.0804,C -0.7402,E1 19.9371,E2 282.6816} C_DIS
LIN {X -124.163,Y 30.6337,Z 150,A 163.136,B 20.0807,C -0.7302,E1 19.9385,E2 284.8306} C_DIS
LIN {X -123.196,Y 34.3098,Z 150,A 161.2865,B 20.0807,C -0.7302,E1 19.9399,E2 286.6937} C_DIS
LIN {X -121.8886,Y 38.699,Z 150,A 160.0543,B 20.0794,C -0.7658,E1 19.9409,E2 287.8307} C_DIS
LIN {X -119.9867,Y 44.2492,Z 150,A 157.2338,B 20.0794,C -0.7668,E1 19.9435,E2 290.6688} C_DIS
LIN {X -119.0239,Y 46.7749,Z 150,A 155.9723,B 20.0794,C -0.7686,E1 19.9447,E2 291.9341} C_DIS
LIN {X -117.6218,Y 50.1978,Z 150,A 154.2287,B 20.0793,C -0.7704,E1 19.9466,E2 293.6848} C_DIS
LIN {X -114.3206,Y 57.3215,Z 150,A 150.7441,B 20.0788,C -0.7817,E1 19.9508,E2 297.1602} C_DIS
LIN {X -112.9078,Y 60.0551,Z 150,A 149.2774,B 20.0788,C -0.7825,E1 19.9527,E2 298.6346} C_DIS
LIN {X -110.997,Y 63.518,Z 150,A 147.1085,B 20.0792,C -0.7732,E1 19.9557,E2 300.8453} C_DIS
LIN {X -109.044,Y 66.815,Z 150,A 145.9265,B 20.0783,C -0.7972,E1 19.9573,E2 301.9646} C_DIS
LIN {X -107.4788,Y 69.3058,Z 150,A 144.3788,B 20.0784,C -0.7925,E1 19.9597,E2 303.5362} C_DIS
LIN {X -105.5756,Y 72.1712,Z 150,A 142.5804,B 20.0786,C -0.7874,E1 19.9625,E2 305.3611} C_DIS
LIN {X -103.6037,Y 74.9742,Z 150,A 141.4952,B 20.0779,C -0.8077,E1 19.9642,E2 306.3935} C_DIS
LIN {X -101.5771,Y 77.6977,Z 150,A 139.6866,B 20.0781,C -0.8012,E1 19.9673,E2 308.2321} C_DIS
LIN {X -98.6492,Y 81.3832,Z 150,A 137.6171,B 20.0779,C -0.808,E1 19.9709,E2 310.294} C_DIS
LIN {X -95.9017,Y 84.6032,Z 150,A 135.7569,B 20.0776,C -0.814,E1 19.9743,E2 312.1474} C_DIS
LIN {X -92.7469,Y 88.0512,Z 150,A 133.5891,B 20.0776,C -0.8163,E1 19.9785,E2 314.3205} C_DIS
LIN {X -89.7954,Y 91.059,Z 150,A 131.783,B 20.0772,C -0.8237,E1 19.982,E2 316.1147} C_DIS
LIN {X -86.8219,Y 93.8985,Z 150,A 129.8346,B 20.0772,C -0.824,E1 19.986,E2 318.0725} C_DIS
LIN {X -84.0415,Y 96.3943,Z 150,A 128.4221,B 20.0767,C -0.8372,E1 19.9889,E2 319.4533} C_DIS
LIN {X -81.7331,Y 98.3594,Z 150,A 126.7926,B 20.077,C -0.8302,E1 19.9924,E2 321.1115} C_DIS
LIN {X -75.3676,Y 103.3185,Z 150,A 123.4642,B 20.0763,C -0.8481,E1 19.9997,E2 324.4029} C_DIS
LIN {X -72.1213,Y 105.6098,Z 150,A 121.3616,B 20.0766,C -0.8395,E1 20.0046,E2 326.5396} C_DIS
LIN {X -68.851,Y 107.7701,Z 150,A 119.6521,B 20.0764,C -0.8445,E1 20.0086,E2 328.2417} C_DIS
LIN {X -66.0787,Y 109.4918,Z 150,A 118.2011,B 20.0763,C -0.8475,E1 20.012,E2 329.6897} C_DIS
LIN {X -62.5883,Y 111.5238,Z 150,A 116.4299,B 20.0761,C -0.852,E1 20.0163,E2 331.4545} C_DIS
LIN {X -59.1157,Y 113.4011,Z 150,A 114.5896,B 20.0761,C -0.8521,E1 20.0208,E2 333.3007} C_DIS
LIN {X -54.8526,Y 115.5233,Z 150,A 112.5603,B 20.0758,C -0.8593,E1 20.0259,E2 335.3159} C_DIS
LIN {X -51.7209,Y 116.9598,Z 150,A 111.0358,B 20.0757,C -0.8622,E1 20.0298,E2 336.8367} C_DIS
LIN {X -48.566,Y 118.306,Z 150,A 109.4587,B 20.0757,C -0.8627,E1 20.0338,E2 338.4168} C_DIS
LIN {X -45.5478,Y 119.5003,Z 150,A 108.0153,B 20.0756,C -0.865,E1 20.0376,E2 339.8576} C_DIS
LIN {X -42.1546,Y 120.7371,Z 150,A 106.1407,B 20.0759,C -0.8573,E1 20.0426,E2 341.7593} C_DIS
LIN {X -38.4204,Y 121.9775,Z 150,A 104.4795,B 20.0757,C -0.863,E1 20.047,E2 343.4075} C_DIS
LIN {X -34.5909,Y 123.1174,Z 150,A 102.781,B 20.0754,C -0.8683,E1 20.0515,E2 345.0941} C_DIS
LIN {X -31.2975,Y 123.9955,Z 150,A 101.2896,B 20.0754,C -0.8711,E1 20.0555,E2 346.5802} C_DIS
LIN {X -28.1344,Y 124.7517,Z 150,A 99.8049,B 20.0754,C -0.8713,E1 20.0596,E2 348.0667} C_DIS
LIN {X -25.4054,Y 125.3355,Z 150,A 97.9055,B 20.0763,C -0.8476,E1 20.065,E2 350.038} C_DIS
LIN {X -20.5981,Y 126.2155,Z 150,A 96.4963,B 20.075,C -0.8788,E1 20.0686,E2 351.3581} C_DIS
LIN {X -18.119,Y 126.5944,Z 150,A 95.2611,B 20.0751,C -0.8752,E1 20.072,E2 352.605} C_DIS
LIN {X -15.1185,Y 126.9877,Z 150,A 93.839,B 20.0752,C -0.8734,E1 20.076,E2 354.0337} C_DIS
LIN {X -10.3431,Y 127.4663,Z 150,A 91.8963,B 20.0749,C -0.8823,E1 20.0813,E2 355.9516} C_DIS
LIN {X -4.7535,Y 127.7965,Z 150,A 89.4734,B 20.0747,C -0.8865,E1 20.0881,E2 358.3633} C_DIS
LIN {X -2.2291,Y 127.8653,Z 150,A 88.0449,B 20.0752,C -0.8752,E1 20.0921,E2 359.825} C_DIS
LIN {X 2.4551,Y 127.8615,Z 150,A 85.7128,B 20.0755,C -0.8663,E1 20.0987,E2 362.1824} C_DIS
LIN {X 7.6454,Y 127.656,Z 150,A 83.6241,B 20.0751,C -0.8756,E1 20.1045,E2 364.2432} C_DIS
LIN {X 11.0553,Y 127.4061,Z 150,A 82.1185,B 20.0751,C -0.8765,E1 20.1086,E2 365.7453} C_DIS
LIN {X 15.1442,Y 126.9846,Z 150,A 80.3027,B 20.0751,C -0.8771,E1 20.1137,E2 367.5575} C_DIS
LIN {X 18.8032,Y 126.4965,Z 150,A 78.6629,B 20.0751,C -0.8771,E1 20.1182,E2 369.1954} C_DIS
LIN {X 21.2444,Y 126.1077,Z 150,A 77.4799,B 20.0752,C -0.8738,E1 20.1215,E2 370.3866} C_DIS
LIN {X 24.6506,Y 125.4878,Z 150,A 75.8522,B 20.0754,C -0.8701,E1 20.126,E2 372.0228} C_DIS
LIN {X 28.392,Y 124.6929,Z 150,A 74.1669,B 20.0754,C -0.8703,E1 20.1306,E2 373.7044} C_DIS
LIN {X 32.7574,Y 123.6179,Z 150,A 72.1659,B 20.0754,C -0.8696,E1 20.136,E2 375.7038} C_DIS
LIN {X 36.7648,Y 122.4876,Z 150,A 70.4392,B 20.0752,C -0.8737,E1 20.1406,E2 377.4147} C_DIS
LIN {X 39.2918,Y 121.6992,Z 150,A 69.2614,B 20.0752,C -0.8731,E1 20.1437,E2 378.5915} C_DIS
LIN {X 42.0317,Y 120.7797,Z 150,A 67.8995,B 20.0754,C -0.8693,E1 20.1473,E2 379.961} C_DIS
LIN {X 45.5072,Y 119.5155,Z 150,A 66.2761,B 20.0754,C -0.8691,E1 20.1515,E2 381.5808} C_DIS
LIN {X 48.8837,Y 118.1733,Z 150,A 64.7907,B 20.0752,C -0.8731,E1 20.1554,E2 383.0501} C_DIS
LIN {X 51.6347,Y 116.9984,Z 150,A 63.3577,B 20.0755,C -0.8679,E1 20.1591,E2 384.4939} C_DIS
LIN {X 54.1057,Y 115.8756,Z 150,A 61.9819,B 20.0758,C -0.86,E1 20.1626,E2 385.8881} C_DIS
LIN {X 58.231,Y 113.8576,Z 150,A 59.9451,B 20.0758,C -0.8582,E1 20.1677,E2 387.923} C_DIS
LIN {X 62.1568,Y 111.765,Z 150,A 57.9166,B 20.076,C -0.8541,E1 20.1727,E2 389.9562} C_DIS
LIN {X 64.8302,Y 110.2356,Z 150,A 56.6033,B 20.076,C -0.8548,E1 20.1758,E2 391.2623} C_DIS
LIN {X 68.5652,Y 107.9527,Z 150,A 54.611,B 20.0762,C -0.8505,E1 20.1805,E2 393.259} C_DIS
LIN {X 72.0011,Y 105.6921,Z 150,A 52.8563,B 20.0762,C -0.8511,E1 20.1846,E2 395.0045} C_DIS
LIN {X 74.2039,Y 104.1569,Z 150,A 51.7239,B 20.0762,C -0.8519,E1 20.1872,E2 396.1293} C_DIS
LIN {X 77.2825,Y 101.8938,Z 150,A 49.8785,B 20.0765,C -0.8435,E1 20.1913,E2 397.9909} C_DIS
LIN {X 80.6823,Y 99.2235,Z 150,A 47.925,B 20.0766,C -0.8392,E1 20.1956,E2 399.9474} C_DIS
LIN {X 83.9406,Y 96.4824,Z 150,A 46.1138,B 20.0766,C -0.8395,E1 20.1994,E2 401.7487} C_DIS
LIN {X 87.4277,Y 93.3347,Z 150,A 44.0853,B 20.0766,C -0.8384,E1 20.2036,E2 403.7698} C_DIS
LIN {X 90.0448,Y 90.8118,Z 150,A 42.5223,B 20.0766,C -0.8378,E1 20.2067,E2 405.3264} C_DIS
LIN {X 92.887,Y 87.9027,Z 150,A 40.5142,B 20.0771,C -0.8261,E1 20.2106,E2 407.3573} C_DIS
LIN {X 95.896,Y 84.6097,Z 150,A 38.5724,B 20.0772,C -0.824,E1 20.2143,E2 409.2942} C_DIS
LIN {X 98.7148,Y 81.3039,Z 150,A 36.6247,B 20.0774,C -0.8195,E1 20.2178,E2 411.2437} C_DIS
LIN {X 101.232,Y 78.1471,Z 150,A 34.831,B 20.0775,C -0.8158,E1 20.2208,E2 413.0373} C_DIS
LIN {X 103.81,Y 74.689,Z 150,A 32.6899,B 20.0781,C -0.8024,E1 20.2244,E2 415.2041} C_DIS
LIN {X 106.5961,Y 70.656,Z 150,A 30.6825,B 20.078,C -0.8047,E1 20.2275,E2 417.192} C_DIS
LIN {X 108.8129,Y 67.1918,Z 150,A 28.785,B 20.0782,C -0.7977,E1 20.2303,E2 419.0977} C_DIS
LIN {X 110.7137,Y 64.0103,Z 150,A 27.3433,B 20.0781,C -0.8025,E1 20.2324,E2 420.5159} C_DIS
LIN {X 112.5244,Y 60.7715,Z 150,A 25.6054,B 20.0784,C -0.7949,E1 20.2347,E2 422.2644} C_DIS
LIN {X 114.0659,Y 57.8219,Z 150,A 24.1804,B 20.0784,C -0.7936,E1 20.2365,E2 423.6833} C_DIS
LIN {X 115.5438,Y 54.8097,Z 150,A 22.6771,B 20.0786,C -0.7895,E1 20.2383,E2 425.1884} C_DIS
LIN {X 117.3254,Y 50.8834,Z 150,A 20.3667,B 20.0794,C -0.7681,E1 20.241,E2 427.5446} C_DIS
LIN {X 118.795,Y 47.3536,Z 150,A 19.1864,B 20.0787,C -0.7857,E1 20.2422,E2 428.6657} C_DIS
LIN {X 119.7913,Y 44.7707,Z 150,A 17.9248,B 20.0789,C -0.7812,E1 20.2434,E2 429.9313} C_DIS
LIN {X 120.7955,Y 41.986,Z 150,A 16.5352,B 20.0791,C -0.7747,E1 20.2447,E2 431.3299} C_DIS
LIN {X 121.8322,Y 38.8754,Z 150,A 15.0626,B 20.0793,C -0.7702,E1 20.246,E2 432.8047} C_DIS
LIN {X 122.8903,Y 35.3933,Z 150,A 13.5001,B 20.0793,C -0.7683,E1 20.2473,E2 434.3616} C_DIS
LIN {X 123.5913,Y 32.8573,Z 150,A 12.2925,B 20.0795,C -0.7635,E1 20.2481,E2 435.574} C_DIS
LIN {X 124.4569,Y 29.4143,Z 150,A 10.7468,B 20.0796,C -0.7606,E1 20.2492,E2 437.1168} C_DIS
LIN {X 125.3576,Y 25.2966,Z 150,A 8.8734,B 20.0798,C -0.7555,E1 20.2503,E2 438.991} C_DIS
LIN {X 126.0248,Y 21.7412,Z 150,A 7.1821,B 20.0801,C -0.7475,E1 20.2511,E2 440.6928} C_DIS
LIN {X 126.7508,Y 16.9951,Z 150,A 4.9301,B 20.0805,C -0.7366,E1 20.252,E2 442.9596} C_DIS
LIN {X 127.3863,Y 11.2897,Z 150,A 2.6681,B 20.0803,C -0.7419,E1 20.2527,E2 445.1893} C_DIS
LIN {X 127.6205,Y 8.2224,Z 150,A 0.548,B 20.0815,C -0.7059,E1 20.2531,E2 447.3972} C_DIS
LIN {X 127.8392,Y 3.4125,Z 150,A -0.9224,B 20.0808,C -0.7284,E1 20.2531,E2 448.7915} C_DIS
LIN {X 127.8823,Y -0.865,Z 150,A -2.864,B 20.081,C -0.7213,E1 20.2532,E2 450.739} C_DIS
LIN {X 127.8082,Y -4.4532,Z 150,A -5.1045,B 20.0821,C -0.6893,E1 20.253,E2 453.0551} C_DIS
LIN {X 127.5456,Y -9.3053,Z 150,A -6.6718,B 20.0815,C -0.7084,E1 20.2527,E2 454.5554} C_DIS
LIN {X 126.983,Y -15.1576,Z 150,A -8.8925,B 20.0811,C -0.7179,E1 20.2521,E2 456.7319} C_DIS
LIN {X 126.4822,Y -18.898,Z 150,A -11.1021,B 20.0821,C -0.6902,E1 20.2512,E2 459.0047} C_DIS
LIN {X 125.9079,Y -22.3972,Z 150,A -12.5574,B 20.0821,C -0.691,E1 20.2506,E2 460.447} C_DIS
LIN {X 125.2239,Y -25.9539,Z 150,A -14.0345,B 20.082,C -0.6922,E1 20.2498,E2 461.9097} C_DIS
LIN {X 124.4844,Y -29.3004,Z 150,A -15.5862,B 20.0822,C -0.6867,E1 20.2488,E2 463.4658} C_DIS
LIN {X 123.504,Y -33.1846,Z 150,A -17.4666,B 20.0825,C -0.6775,E1 20.2475,E2 465.359} C_DIS
LIN {X 122.3049,Y -37.3618,Z 150,A -19.243,B 20.0825,C -0.6788,E1 20.2461,E2 467.1186} C_DIS
LIN {X 121.2745,Y -40.5822,Z 150,A -20.8559,B 20.0827,C -0.67,E1 20.2447,E2 468.7453} C_DIS
LIN {X 119.7315,Y -44.9303,Z 150,A -22.8978,B 20.0829,C -0.6649,E1 20.2427,E2 470.7876} C_DIS
LIN {X 118.3067,Y -48.5642,Z 150,A -24.5925,B 20.0829,C -0.6619,E1 20.241,E2 472.4789} C_DIS
LIN {X 117.23,Y -51.1041,Z 150,A -25.8005,B 20.0831,C -0.6595,E1 20.2396,E2 473.6855} C_DIS
LIN {X 115.7891,Y -54.2928,Z 150,A -27.3864,B 20.0832,C -0.6541,E1 20.2378,E2 475.2761} C_DIS
LIN {X 113.8294,Y -58.2864,Z 150,A -29.3583,B 20.0834,C -0.6492,E1 20.2353,E2 477.2486} C_DIS
LIN {X 112.2145,Y -61.3413,Z 150,A -30.9281,B 20.0835,C -0.6439,E1 20.2333,E2 478.8234} C_DIS
LIN {X 109.6851,Y -65.7581,Z 150,A -33.2987,B 20.0839,C -0.6336,E1 20.2299,E2 481.2082} C_DIS
LIN {X 107.3172,Y -69.5548,Z 150,A -35.1243,B 20.0838,C -0.6357,E1 20.2272,E2 483.016} C_DIS
LIN {X 105.3091,Y -72.5596,Z 150,A -36.8662,B 20.0841,C -0.6261,E1 20.2244,E2 484.7747} C_DIS
LIN {X 102.9596,Y -75.8563,Z 150,A -38.7864,B 20.0844,C -0.6168,E1 20.2213,E2 486.7101} C_DIS
LIN {X 100.1371,Y -79.545,Z 150,A -40.58,B 20.0842,C -0.6236,E1 20.2183,E2 488.4733} C_DIS
LIN {X 97.7431,Y -82.4696,Z 150,A -42.4039,B 20.0844,C -0.6137,E1 20.215,E2 490.3149} C_DIS
LIN {X 94.1785,Y -86.5174,Z 150,A -45.3907,B 20.0853,C -0.5838,E1 20.2092,E2 493.3714} C_DIS
LIN {X 90.7287,Y -90.1284,Z 150,A -46.9232,B 20.0846,C -0.6081,E1 20.2064,E2 494.8253} C_DIS
LIN {X 88.0068,Y -92.7888,Z 150,A -49.1996,B 20.0854,C -0.5802,E1 20.2017,E2 497.1705} C_DIS
LIN {X 84.7489,Y -95.773,Z 150,A -50.7942,B 20.0851,C -0.5918,E1 20.1984,E2 498.7232} C_DIS
LIN {X 82.1811,Y -97.9852,Z 150,A -52.1033,B 20.0849,C -0.5973,E1 20.1957,E2 500.0101} C_DIS
LIN {X 79.2602,Y -100.3632,Z 150,A -53.9301,B 20.0852,C -0.5879,E1 20.1917,E2 501.8554} C_DIS
LIN {X 74.9944,Y -103.589,Z 150,A -56.1697,B 20.0852,C -0.5896,E1 20.1867,E2 504.0798} C_DIS
LIN {X 73.0052,Y -105.0003,Z 150,A -57.3734,B 20.0853,C -0.5828,E1 20.1839,E2 505.2979} C_DIS
LIN {X 69.2995,Y -107.4829,Z 150,A -59.394,B 20.0855,C -0.5781,E1 20.1792,E2 507.3236} C_DIS
LIN {X 63.51,Y -111.0015,Z 150,A -62.2673,B 20.0855,C -0.5795,E1 20.1723,E2 510.1816} C_DIS
LIN {X 60.9445,Y -112.431,Z 150,A -63.7416,B 20.0857,C -0.5707,E1 20.1687,E2 511.676} C_DIS
LIN {X 57.7169,Y -114.1193,Z 150,A -65.1611,B 20.0855,C -0.5769,E1 20.1652,E2 513.0725} C_DIS
LIN {X 54.9455,Y -115.4789,Z 150,A -66.697,B 20.0857,C -0.5684,E1 20.1613,E2 514.6277} C_DIS
LIN {X 48.4825,Y -118.3399,Z 150,A -69.7061,B 20.0857,C -0.5703,E1 20.1536,E2 517.622} C_DIS
LIN {X 45.7281,Y -119.4308,Z 150,A -71.1682,B 20.0859,C -0.5631,E1 20.1498,E2 519.1011} C_DIS
LIN {X 40.5714,Y -121.2781,Z 150,A -73.5664,B 20.0859,C -0.5624,E1 20.1435,E2 521.4951} C_DIS
LIN {X 37.041,Y -122.4031,Z 150,A -75.154,B 20.0859,C -0.5635,E1 20.1392,E2 523.0758} C_DIS
LIN {X 33.4801,Y -123.4252,Z 150,A -77.0617,B 20.0862,C -0.5517,E1 20.134,E2 525.0139} C_DIS
LIN {X 28.0136,Y -124.7793,Z 150,A -79.2736,B 20.0859,C -0.562,E1 20.1281,E2 527.1916} C_DIS
LIN {X 24.7434,Y -125.4701,Z 150,A -80.8055,B 20.0859,C -0.5594,E1 20.1239,E2 528.7288} C_DIS
LIN {X 22.2962,Y -125.926,Z 150,A -82.0891,B 20.0862,C -0.5517,E1 20.1203,E2 530.0328} C_DIS
LIN {X 16.8308,Y -126.7723,Z 150,A -84.785,B 20.0864,C -0.5414,E1 20.1128,E2 532.7557} C_DIS
LIN {X 13.3985,Y -127.181,Z 150,A -86.0238,B 20.0861,C -0.553,E1 20.1095,E2 533.9596} C_DIS
LIN {X 5.3804,Y -127.772,Z 150,A -89.3983,B 20.0859,C -0.5606,E1 20.1001,E2 537.3099} C_DIS
LIN {X 0.9061,Y -127.8608,Z 150,A -90.7259,B 20.0852,C -0.5876,E1 20.0967,E2 538.5585} C_DIS
Enddeposition()
LIN {X 0.9061,Y -127.8608,Z 150,A -90.7259,B 20.0852,C -0.5876,E1 20.0967,E2 538.5585} C_DIS
Startdeposition()
$VEL.CP = VEL_PRINT
LIN {X 1.8372,Y -126.9247,Z 150,A -90.1553,B 18.8945,C -0.4348,E1 18.9032,E2 538.3263} C_DIS
LIN {X 4.9256,Y -126.842,Z 150,A -88.7622,B 18.8945,C -0.4352,E1 18.907,E2 536.9326} C_DIS
LIN {X 7.7668,Y -126.6998,Z 150,A -87.4863,B 18.8945,C -0.4353,E1 18.9106,E2 535.6569} C_DIS
LIN {X 11.1944,Y -126.444,Z 150,A -85.9273,B 18.8945,C -0.4363,E1 18.9149,E2 534.0961} C_DIS
LIN {X 14.2715,Y -126.1346,Z 150,A -84.5622,B 18.8945,C -0.4358,E1 18.9187,E2 532.7337} C_DIS
LIN {X 17.3377,Y -125.7494,Z 150,A -83.1413,B 18.8945,C -0.4376,E1 18.9227,E2 531.3088} C_DIS
LIN {X 20.3964,Y -125.2891,Z 150,A -81.8303,B 18.8945,C -0.4353,E1 18.9263,E2 530.0067} C_DIS
LIN {X 23.5327,Y -124.7374,Z 150,A -80.3169,B 18.8945,C -0.4393,E1 18.9304,E2 528.4834} C_DIS
LIN {X 26.2846,Y -124.1873,Z 150,A -78.9703,B 18.8943,C -0.4434,E1 18.9342,E2 527.1265} C_DIS
LIN {X 29.6119,Y -123.4352,Z 150,A -77.6056,B 18.8944,C -0.438,E1 18.9378,E2 525.7809} C_DIS
LIN {X 32.337,Y -122.7499,Z 150,A -76.164,B 18.8943,C -0.4459,E1 18.9418,E2 524.3181} C_DIS
LIN {X 35.3556,Y -121.9146,Z 150,A -74.7735,B 18.8943,C -0.4464,E1 18.9455,E2 522.929} C_DIS
LIN {X 38.3326,Y -121.0115,Z 150,A -73.4455,B 18.8943,C -0.445,E1 18.949,E2 521.6087} C_DIS
LIN {X 41.595,Y -119.9288,Z 150,A -71.9002,B 18.8943,C -0.4466,E1 18.9531,E2 520.0626} C_DIS
LIN {X 45.0855,Y -118.6622,Z 150,A -70.0115,B 18.894,C -0.457,E1 18.9581,E2 518.1474} C_DIS
LIN {X 49.01,Y -117.0943,Z 150,A -68.4574,B 18.8943,C -0.4458,E1 18.962,E2 516.6327} C_DIS
LIN {X 51.4148,Y -116.0593,Z 150,A -67.1468,B 18.8941,C -0.4525,E1 18.9654,E2 515.3058} C_DIS
LIN {X 54.2679,Y -114.7531,Z 150,A -65.7435,B 18.8941,C -0.454,E1 18.969,E2 513.9027} C_DIS
LIN {X 57.3433,Y -113.2468,Z 150,A -64.2054,B 18.8941,C -0.4562,E1 18.9728,E2 512.3637} C_DIS
LIN {X 60.102,Y -111.8091,Z 150,A -62.8738,B 18.8941,C -0.4556,E1 18.9761,E2 511.0391} C_DIS
LIN {X 62.556,Y -110.4555,Z 150,A -61.5445,B 18.8939,C -0.4602,E1 18.9794,E2 509.7008} C_DIS
LIN {X 65.1867,Y -108.9232,Z 150,A -60.1607,B 18.8939,C -0.463,E1 18.9827,E2 508.3143} C_DIS
LIN {X 68.1674,Y -107.0833,Z 150,A -58.611,B 18.8939,C -0.4646,E1 18.9864,E2 506.7663} C_DIS
LIN {X 70.8443,Y -105.3316,Z 150,A -57.1772,B 18.8938,C -0.4669,E1 18.9897,E2 505.3321} C_DIS
LIN {X 73.0811,Y -103.7916,Z 150,A -55.9515,B 18.8938,C -0.4692,E1 18.9925,E2 504.1048} C_DIS
LIN {X 75.6273,Y -101.9514,Z 150,A -54.4173,B 18.8935,C -0.4767,E1 18.996,E2 502.5552} C_DIS
LIN {X 78.7071,Y -99.5934,Z 150,A -52.6343,B 18.8935,C -0.4815,E1 18.9999,E2 500.7662} C_DIS
LIN {X 82.3048,Y -96.6409,Z 150,A -50.5863,B 18.8934,C -0.4839,E1 19.0043,E2 498.7216} C_DIS
LIN {X 85.327,Y -93.9831,Z 150,A -48.7697,B 18.8933,C -0.4879,E1 19.0081,E2 496.9026} C_DIS
LIN {X 88.5391,Y -90.9641,Z 150,A -46.8618,B 18.8933,C -0.4892,E1 19.0119,E2 495.0016} C_DIS
LIN {X 91.3785,Y -88.1111,Z 150,A -44.9911,B 18.8931,C -0.4956,E1 19.0156,E2 493.1221} C_DIS
LIN {X 94.0202,Y -85.2861,Z 150,A -43.3456,B 18.8931,C -0.4958,E1 19.0187,E2 491.4859} C_DIS
LIN {X 96.6265,Y -82.3216,Z 150,A -41.4656,B 18.8928,C -0.5042,E1 19.0222,E2 489.5918} C_DIS
LIN {X 99.5821,Y -78.7216,Z 150,A -39.3672,B 18.8928,C -0.5093,E1 19.0258,E2 487.491} C_DIS
LIN {X 102.1437,Y -75.3674,Z 150,A -37.6432,B 18.8928,C -0.507,E1 19.0287,E2 485.7853} C_DIS
LIN {X 103.7844,Y -73.0913,Z 150,A -36.3293,B 18.8926,C -0.5122,E1 19.0308,E2 484.464} C_DIS
LIN {X 105.5442,Y -70.5263,Z 150,A -34.9878,B 18.8926,C -0.5135,E1 19.0329,E2 483.1278} C_DIS
LIN {X 107.41,Y -67.6508,Z 150,A -33.4501,B 18.8926,C -0.5173,E1 19.0352,E2 481.5888} C_DIS
LIN {X 109.0287,Y -65.0098,Z 150,A -32.0652,B 18.8924,C -0.5206,E1 19.0372,E2 480.2034} C_DIS
LIN {X 110.5969,Y -62.3047,Z 150,A -30.7001,B 18.8924,C -0.5226,E1 19.0391,E2 478.8416} C_DIS
LIN {X 111.954,Y -59.8322,Z 150,A -29.3751,B 18.8922,C -0.5283,E1 19.0409,E2 477.5086} C_DIS
LIN {X 113.5304,Y -56.7835,Z 150,A -27.871,B 18.8922,C -0.5309,E1 19.0428,E2 476.0075} C_DIS
LIN {X 114.8864,Y -53.9886,Z 150,A -26.4683,B 18.892,C -0.535,E1 19.0445,E2 474.6025} C_DIS
LIN {X 116.3311,Y -50.7969,Z 150,A -25.03,B 18.892,C -0.5338,E1 19.0461,E2 473.1785} C_DIS
LIN {X 117.2736,Y -48.5807,Z 150,A -23.8221,B 18.8918,C -0.5419,E1 19.0474,E2 471.9549} C_DIS
LIN {X 118.4283,Y -45.6935,Z 150,A -22.4309,B 18.8918,C -0.5456,E1 19.0488,E2 470.5629} C_DIS
LIN {X 119.5117,Y -42.7797,Z 150,A -20.9101,B 18.8915,C -0.5545,E1 19.0503,E2 469.0262} C_DIS
LIN {X 120.6266,Y -39.5304,Z 150,A -19.5194,B 18.8915,C -0.5527,E1 19.0515,E2 467.6519} C_DIS
LIN {X 121.5648,Y -36.544,Z 150,A -18.1031,B 18.8915,C -0.5571,E1 19.0527,E2 466.233} C_DIS
LIN {X 122.4236,Y -33.5556,Z 150,A -16.7131,B 18.8913,C -0.5608,E1 19.0537,E2 464.8425} C_DIS
LIN {X 123.1342,Y -30.8416,Z 150,A -15.4215,B 18.8912,C -0.5657,E1 19.0546,E2 463.546} C_DIS
LIN {X 123.9206,Y -27.5201,Z 150,A -13.9369,B 18.8912,C -0.5681,E1 19.0556,E2 462.0656} C_DIS
LIN {X 124.4981,Y -24.7715,Z 150,A -12.6149,B 18.8909,C -0.5743,E1 19.0563,E2 460.7353} C_DIS
LIN {X 125.068,Y -21.7148,Z 150,A -11.2177,B 18.8909,C -0.5783,E1 19.057,E2 459.3367} C_DIS
LIN {X 125.6161,Y -18.2708,Z 150,A -9.7207,B 18.8907,C -0.5801,E1 19.0576,E2 457.8464} C_DIS
LIN {X 125.9831,Y -15.5456,Z 150,A -8.3994,B 18.8905,C -0.5872,E1 19.0581,E2 456.5139} C_DIS
LIN {X 126.3274,Y -12.4353,Z 150,A -7.0167,B 18.8905,C -0.5904,E1 19.0585,E2 455.1325} C_DIS
LIN {X 126.6152,Y -9.0435,Z 150,A -5.6176,B 18.8905,C -0.5896,E1 19.0588,E2 453.7471} C_DIS
LIN {X 126.8006,Y -5.9139,Z 150,A -4.2001,B 18.8903,C -0.5941,E1 19.059,E2 452.3273} C_DIS
LIN {X 126.9,Y -3.1186,Z 150,A -2.833,B 18.8901,C -0.6023,E1 19.059,E2 450.9462} C_DIS
LIN {X 126.9401,Y -0.0217,Z 150,A -1.4034,B 18.8899,C -0.6079,E1 19.0591,E2 449.511} C_DIS
LIN {X 126.8928,Y 3.3764,Z 150,A -0.073,B 18.89,C -0.6044,E1 19.0591,E2 448.202} C_DIS
LIN {X 126.7689,Y 6.5446,Z 150,A 1.362,B 18.8899,C -0.609,E1 19.0589,E2 446.7645} C_DIS
LIN {X 126.5889,Y 9.4041,Z 150,A 2.7219,B 18.8897,C -0.6157,E1 19.0586,E2 445.3951} C_DIS
LIN {X 126.3283,Y 12.4254,Z 150,A 4.0753,B 18.8896,C -0.6193,E1 19.0582,E2 444.0415} C_DIS
LIN {X 125.9883,Y 15.5014,Z 150,A 5.4767,B 18.8894,C -0.6238,E1 19.0578,E2 442.6377} C_DIS
LIN {X 125.5184,Y 18.9341,Z 150,A 7.0019,B 18.8894,C -0.627,E1 19.0572,E2 441.1149} C_DIS
LIN {X 125.0705,Y 21.7008,Z 150,A 8.3476,B 18.8891,C -0.6341,E1 19.0566,E2 439.7581} C_DIS
LIN {X 124.4412,Y 25.0514,Z 150,A 9.682,B 18.8891,C -0.6305,E1 19.0559,E2 438.4453} C_DIS
LIN {X 123.7864,Y 28.108,Z 150,A 11.178,B 18.8889,C -0.6382,E1 19.0549,E2 436.9376} C_DIS
LIN {X 123.1326,Y 30.8482,Z 150,A 12.438,B 18.8889,C -0.6415,E1 19.0541,E2 435.6774} C_DIS
LIN {X 122.3396,Y 33.856,Z 150,A 13.83,B 18.8887,C -0.6452,E1 19.0531,E2 434.285} C_DIS
LIN {X 121.3834,Y 37.1368,Z 150,A 15.468,B 18.8884,C -0.6535,E1 19.0518,E2 432.634} C_DIS
LIN {X 120.0322,Y 41.2967,Z 150,A 17.3877,B 18.8884,C -0.6571,E1 19.0501,E2 430.7182} C_DIS
LIN {X 118.6729,Y 45.0569,Z 150,A 19.258,B 18.8881,C -0.6649,E1 19.0482,E2 428.8383} C_DIS
LIN {X 117.2879,Y 48.5463,Z 150,A 20.7979,B 18.8881,C -0.6634,E1 19.0466,E2 427.3143} C_DIS
LIN {X 116.0476,Y 51.4411,Z 150,A 22.1955,B 18.8881,C -0.6664,E1 19.0451,E2 425.9178} C_DIS
LIN {X 114.7528,Y 54.2686,Z 150,A 23.5866,B 18.8879,C -0.6698,E1 19.0434,E2 424.5266} C_DIS
LIN {X 113.2465,Y 57.3441,Z 150,A 25.1691,B 18.8877,C -0.6755,E1 19.0415,E2 422.9382} C_DIS
LIN {X 111.8046,Y 60.1104,Z 150,A 26.4464,B 18.8877,C -0.674,E1 19.0398,E2 421.6746} C_DIS
LIN {X 110.4482,Y 62.5688,Z 150,A 27.7832,B 18.8875,C -0.6801,E1 19.038,E2 420.3285} C_DIS
LIN {X 108.8727,Y 65.2715,Z 150,A 29.1902,B 18.8875,C -0.6836,E1 19.036,E2 418.9208} C_DIS
LIN {X 107.0818,Y 68.1698,Z 150,A 30.7039,B 18.8873,C -0.6866,E1 19.0337,E2 417.4083} C_DIS
LIN {X 105.5507,Y 70.5164,Z 150,A 32.0193,B 18.8871,C -0.6918,E1 19.0317,E2 416.0859} C_DIS
LIN {X 103.7951,Y 73.0761,Z 150,A 33.3612,B 18.8871,C -0.6929,E1 19.0296,E2 414.7495} C_DIS
LIN {X 101.7226,Y 75.9346,Z 150,A 35.0513,B 18.8868,C -0.7005,E1 19.0267,E2 413.0469} C_DIS
LIN {X 99.1013,Y 79.3257,Z 150,A 36.8909,B 18.8868,C -0.7013,E1 19.0236,E2 411.2167} C_DIS
LIN {X 96.6249,Y 82.3235,Z 150,A 38.7339,B 18.8865,C -0.7088,E1 19.0203,E2 409.3622} C_DIS
LIN {X 93.7124,Y 85.625,Z 150,A 40.6479,B 18.8865,C -0.7103,E1 19.0167,E2 407.4551} C_DIS
LIN {X 90.8504,Y 88.6557,Z 150,A 42.5714,B 18.8863,C -0.716,E1 19.013,E2 405.5254} C_DIS
LIN {X 88.0959,Y 91.3932,Z 150,A 44.3291,B 18.8861,C -0.7198,E1 19.0095,E2 403.766} C_DIS
LIN {X 85.0358,Y 94.2473,Z 150,A 46.2163,B 18.886,C -0.7235,E1 19.0056,E2 401.8779} C_DIS
LIN {X 81.7291,Y 97.1283,Z 150,A 48.1614,B 18.8859,C -0.726,E1 19.0014,E2 399.9356} C_DIS
LIN {X 78.5968,Y 99.6801,Z 150,A 49.9818,B 18.8858,C -0.7292,E1 18.9975,E2 398.1146} C_DIS
LIN {X 75.1346,Y 102.3148,Z 150,A 51.7364,B 18.8859,C -0.7245,E1 18.9936,E2 396.383} C_DIS
LIN {X 72.9473,Y 103.8859,Z 150,A 53.0463,B 18.8857,C -0.7302,E1 18.9906,E2 395.0619} C_DIS
LIN {X 70.5184,Y 105.5494,Z 150,A 54.3697,B 18.8857,C -0.7322,E1 18.9875,E2 393.7386} C_DIS
LIN {X 67.6573,Y 107.4059,Z 150,A 55.8795,B 18.8857,C -0.7334,E1 18.984,E2 392.2316} C_DIS
LIN {X 65.009,Y 109.0292,Z 150,A 57.2762,B 18.8855,C -0.7353,E1 18.9806,E2 390.835} C_DIS
LIN {X 62.3228,Y 110.5867,Z 150,A 58.7945,B 18.8853,C -0.7418,E1 18.9769,E2 389.303} C_DIS
LIN {X 58.4616,Y 112.675,Z 150,A 60.8026,B 18.8852,C -0.7454,E1 18.972,E2 387.2913} C_DIS
LIN {X 55.399,Y 114.2128,Z 150,A 62.1783,B 18.8853,C -0.7408,E1 18.9686,E2 385.9349} C_DIS
LIN {X 52.585,Y 115.5354,Z 150,A 63.6703,B 18.8851,C -0.7458,E1 18.9648,E2 384.4326} C_DIS
LIN {X 49.739,Y 116.7885,Z 150,A 64.9796,B 18.8852,C -0.7438,E1 18.9614,E2 383.1338} C_DIS
LIN {X 47.1339,Y 117.8625,Z 150,A 66.2541,B 18.8852,C -0.7452,E1 18.9581,E2 381.8589} C_DIS
LIN {X 44.2368,Y 118.98,Z 150,A 67.6525,B 18.8852,C -0.7465,E1 18.9545,E2 380.4608} C_DIS
LIN {X 40.5743,Y 120.279,Z 150,A 69.2866,B 18.8852,C -0.7435,E1 18.9502,E2 378.8403} C_DIS
LIN {X 38.3322,Y 121.0116,Z 150,A 70.4925,B 18.885,C -0.7497,E1 18.947,E2 377.6183} C_DIS
LIN {X 35.0646,Y 121.9998,Z 150,A 71.9979,B 18.885,C -0.7495,E1 18.9429,E2 376.1172} C_DIS
LIN {X 31.6636,Y 122.9256,Z 150,A 73.7312,B 18.8848,C -0.7559,E1 18.9382,E2 374.3677} C_DIS
LIN {X 27.5062,Y 123.9236,Z 150,A 75.4985,B 18.885,C -0.7509,E1 18.9335,E2 372.6193} C_DIS
LIN {X 24.7624,Y 124.5,Z 150,A 76.8366,B 18.8848,C -0.7542,E1 18.9298,E2 371.2731} C_DIS
LIN {X 20.1728,Y 125.3264,Z 150,A 78.8888,B 18.8848,C -0.7531,E1 18.9241,E2 369.2275} C_DIS
LIN {X 16.7972,Y 125.8216,Z 150,A 80.3307,B 18.885,C -0.7499,E1 18.9202,E2 367.797} C_DIS
LIN {X 13.6827,Y 126.198,Z 150,A 81.7592,B 18.885,C -0.7507,E1 18.9162,E2 366.3675} C_DIS
LIN {X 10.5911,Y 126.495,Z 150,A 83.2321,B 18.8848,C -0.7536,E1 18.9121,E2 364.8871} C_DIS
LIN {X 7.7932,Y 126.6982,Z 150,A 84.5428,B 18.8848,C -0.7553,E1 18.9084,E2 363.5719} C_DIS
LIN {X 4.6912,Y 126.8512,Z 150,A 85.8928,B 18.8848,C -0.7534,E1 18.9047,E2 362.2283} C_DIS
LIN {X 1.2946,Y 126.9325,Z 150,A 87.3876,B 18.8849,C -0.7518,E1 18.9005,E2 360.7387} C_DIS
LIN {X -1.8579,Y 126.9243,Z 150,A 88.8694,B 18.8849,C -0.7537,E1 18.8964,E2 359.251} C_DIS
LIN {X -4.6617,Y 126.8523,Z 150,A 90.1971,B 18.8848,C -0.7557,E1 18.8927,E2 357.9169} C_DIS
LIN {X -8.2681,Y 126.6689,Z 150,A 91.9341,B 18.8846,C -0.7591,E1 18.8878,E2 356.1687} C_DIS
LIN {X -12.4461,Y 126.3263,Z 150,A 93.6722,B 18.8849,C -0.7527,E1 18.883,E2 354.4493} C_DIS
LIN {X -15.5349,Y 125.9843,Z 150,A 95.167,B 18.8848,C -0.7553,E1 18.8788,E2 352.9449} C_DIS
LIN {X -18.9103,Y 125.5221,Z 150,A 96.6085,B 18.8849,C -0.751,E1 18.8749,E2 351.5154} C_DIS
LIN {X -21.6774,Y 125.0747,Z 150,A 97.9702,B 18.8849,C -0.7536,E1 18.8711,E2 350.1437} C_DIS
LIN {X -25.4869,Y 124.3525,Z 150,A 99.6757,B 18.8849,C -0.7507,E1 18.8664,E2 348.4445} C_DIS
LIN {X -29.62,Y 123.4332,Z 150,A 101.4528,B 18.8852,C -0.7444,E1 18.8617,E2 346.6841} C_DIS
LIN {X -32.344,Y 122.7481,Z 150,A 102.8107,B 18.8852,C -0.7464,E1 18.858,E2 345.317} C_DIS
LIN {X -35.7086,Y 121.8112,Z 150,A 104.3769,B 18.8852,C -0.7445,E1 18.8538,E2 343.7533} C_DIS
LIN {X -38.3347,Y 121.0108,Z 150,A 105.637,B 18.8852,C -0.744,E1 18.8504,E2 342.492} C_DIS
LIN {X -41.5921,Y 119.9298,Z 150,A 107.186,B 18.8852,C -0.7422,E1 18.8463,E2 340.9444} C_DIS
LIN {X -44.5169,Y 118.8751,Z 150,A 108.5941,B 18.8853,C -0.7407,E1 18.8426,E2 339.5371} C_DIS
LIN {X -47.5446,Y 117.6969,Z 150,A 109.9523,B 18.8856,C -0.735,E1 18.8391,E2 338.1925} C_DIS
LIN {X -50.0079,Y 116.6723,Z 150,A 111.2711,B 18.8855,C -0.7374,E1 18.8357,E2 336.8622} C_DIS
LIN {X -52.851,Y 115.4124,Z 150,A 112.6785,B 18.8855,C -0.7356,E1 18.8321,E2 335.4557} C_DIS
LIN {X -55.6631,Y 114.0831,Z 150,A 114.1825,B 18.8855,C -0.7371,E1 18.8283,E2 333.942} C_DIS
LIN {X -58.7431,Y 112.5272,Z 150,A 115.6038,B 18.8857,C -0.7299,E1 18.8248,E2 332.5377} C_DIS
LIN {X -61.2154,Y 111.2038,Z 150,A 116.9232,B 18.8857,C -0.7297,E1 18.8216,E2 331.2138} C_DIS
LIN {X -63.9185,Y 109.6726,Z 150,A 118.3429,B 18.8858,C -0.728,E1 18.8181,E2 329.7937} C_DIS
LIN {X -66.5833,Y 108.0752,Z 150,A 119.8068,B 18.8858,C -0.7277,E1 18.8146,E2 328.3244} C_DIS
LIN {X -69.4798,Y 106.2366,Z 150,A 121.265,B 18.886,C -0.7218,E1 18.8112,E2 326.8782} C_DIS
LIN {X -72.0596,Y 104.5037,Z 150,A 122.7404,B 18.886,C -0.7218,E1 18.8078,E2 325.3964} C_DIS
LIN {X -74.7662,Y 102.5849,Z 150,A 124.1213,B 18.8863,C -0.7148,E1 18.8047,E2 324.0304} C_DIS
LIN {X -77.4332,Y 100.5872,Z 150,A 125.8928,B 18.8861,C -0.7211,E1 18.8007,E2 322.2307} C_DIS
LIN {X -80.6447,Y 98.0312,Z 150,A 127.7357,B 18.8862,C -0.7169,E1 18.7967,E2 320.3913} C_DIS
LIN {X -83.9646,Y 95.2023,Z 150,A 129.643,B 18.8865,C -0.7106,E1 18.7927,E2 318.4934} C_DIS
LIN {X -86.9673,Y 92.4675,Z 150,A 131.5721,B 18.8865,C -0.7098,E1 18.7888,E2 316.556} C_DIS
LIN {X -90.3063,Y 89.21,Z 150,A 133.678,B 18.8867,C -0.705,E1 18.7846,E2 314.453} C_DIS
LIN {X -93.362,Y 86.0063,Z 150,A 135.6321,B 18.8869,C -0.6988,E1 18.7809,E2 312.5065} C_DIS
LIN {X -96.1212,Y 82.9111,Z 150,A 137.5713,B 18.8869,C -0.6966,E1 18.7773,E2 310.5624} C_DIS
LIN {X -98.7113,Y 79.81,Z 150,A 139.3888,B 18.8871,C -0.6918,E1 18.7741,E2 308.7482} C_DIS
LIN {X -101.2075,Y 76.6198,Z 150,A 141.1057,B 18.8874,C -0.6834,E1 18.7712,E2 307.0464} C_DIS
LIN {X -103.2866,Y 73.793,Z 150,A 142.8056,B 18.8874,C -0.6832,E1 18.7684,E2 305.3358} C_DIS
LIN {X -105.5505,Y 70.5167,Z 150,A 144.5171,B 18.8877,C -0.6755,E1 18.7657,E2 303.6366} C_DIS
LIN {X -107.4089,Y 67.6526,Z 150,A 146.0794,B 18.8878,C -0.6721,E1 18.7634,E2 302.0742} C_DIS
LIN {X -109.0489,Y 64.9758,Z 150,A 147.4976,B 18.8879,C -0.6683,E1 18.7613,E2 300.658} C_DIS
LIN {X -110.6025,Y 62.2947,Z 150,A 148.9256,B 18.888,C -0.6654,E1 18.7593,E2 299.2287} C_DIS
LIN {X -111.9489,Y 59.8418,Z 150,A 150.276,B 18.888,C -0.6648,E1 18.7575,E2 297.8703} C_DIS
LIN {X -113.5115,Y 56.8218,Z 150,A 151.7162,B 18.8883,C -0.6572,E1 18.7557,E2 296.4431} C_DIS
LIN {X -114.8632,Y 54.0375,Z 150,A 153.1435,B 18.8884,C -0.6543,E1 18.754,E2 295.0145} C_DIS
LIN {X -116.3406,Y 50.775,Z 150,A 154.6263,B 18.8887,C -0.6451,E1 18.7523,E2 293.5491} C_DIS
LIN {X -117.2752,Y 48.5769,Z 150,A 155.8551,B 18.8887,C -0.647,E1 18.751,E2 292.305} C_DIS
LIN {X -118.4302,Y 45.6887,Z 150,A 157.2699,B 18.8887,C -0.6433,E1 18.7496,E2 290.8911} C_DIS
LIN {X -119.7139,Y 42.2148,Z 150,A 158.9113,B 18.889,C -0.6373,E1 18.748,E2 289.2557} C_DIS
LIN {X -120.6256,Y 39.5335,Z 150,A 160.2251,B 18.889,C -0.6346,E1 18.7468,E2 287.9398} C_DIS
LIN {X -121.553,Y 36.5827,Z 150,A 161.6488,B 18.8892,C -0.6314,E1 18.7457,E2 286.5152} C_DIS
LIN {X -122.4067,Y 33.6161,Z 150,A 163.0521,B 18.8892,C -0.6275,E1 18.7446,E2 285.1129} C_DIS
LIN {X -123.1194,Y 30.9001,Z 150,A 164.4417,B 18.8892,C -0.6278,E1 18.7436,E2 283.7114} C_DIS
LIN {X -123.9208,Y 27.519,Z 150,A 165.9048,B 18.8895,C -0.6194,E1 18.7427,E2 282.2626} C_DIS
LIN {X -124.5388,Y 24.5717,Z 150,A 167.3396,B 18.8895,C -0.6178,E1 18.7419,E2 280.8213} C_DIS
LIN {X -125.0713,Y 21.6963,Z 150,A 168.6606,B 18.8897,C -0.6137,E1 18.7413,E2 279.5021} C_DIS
LIN {X -125.5655,Y 18.6251,Z 150,A 170.1374,B 18.8897,C -0.6118,E1 18.7407,E2 278.0192} C_DIS
LIN {X -125.9835,Y 15.5421,Z 150,A 171.5426,B 18.8899,C -0.6075,E1 18.7402,E2 276.616} C_DIS
LIN {X -126.3268,Y 12.4408,Z 150,A 172.9456,B 18.8901,C -0.603,E1 18.7398,E2 275.2156} C_DIS
LIN {X -126.6163,Y 9.0278,Z 150,A 174.376,B 18.8903,C -0.5943,E1 18.7395,E2 273.8005} C_DIS
LIN {X -126.8002,Y 5.923,Z 150,A 175.806,B 18.8904,C -0.5908,E1 18.7393,E2 272.3697} C_DIS
LIN {X -126.9006,Y 3.0965,Z 150,A 177.2182,B 18.8904,C -0.5914,E1 18.7391,E2 270.944} C_DIS
LIN {X -126.9402,Y -0.0154,Z 150,A 178.6771,B 18.8904,C -0.5888,E1 18.7391,E2 269.4811} C_DIS
LIN {X -126.8758,Y -3.9902,Z 150,A -179.4784,B 18.8906,C -0.585,E1 18.7393,E2 267.6334} C_DIS
LIN {X -126.6987,Y -7.7837,Z 150,A -177.8854,B 18.8909,C -0.5756,E1 18.7395,E2 266.0565} C_DIS
LIN {X -126.4447,Y -11.1866,Z 150,A -176.3895,B 18.8911,C -0.5694,E1 18.7398,E2 264.5678} C_DIS
LIN {X -126.1339,Y -14.2784,Z 150,A -174.8073,B 18.8911,C -0.5711,E1 18.7403,E2 262.9672} C_DIS
LIN {X -125.7422,Y -17.3887,Z 150,A -173.5021,B 18.8912,C -0.5631,E1 18.7408,E2 261.6764} C_DIS
LIN {X -125.2774,Y -20.4664,Z 150,A -172.2006,B 18.8915,C -0.5553,E1 18.7414,E2 260.3885} C_DIS
LIN {X -124.7383,Y -23.5282,Z 150,A -170.6747,B 18.8915,C -0.5553,E1 18.7421,E2 258.8505} C_DIS
LIN {X -124.0874,Y -26.7472,Z 150,A -169.2212,B 18.8916,C -0.5498,E1 18.7429,E2 257.4022} C_DIS
LIN {X -123.4315,Y -29.6273,Z 150,A -167.9261,B 18.8918,C -0.5445,E1 18.7438,E2 256.1132} C_DIS
LIN {X -122.7462,Y -32.3511,Z 150,A -166.5603,B 18.8918,C -0.5441,E1 18.7447,E2 254.7379} C_DIS
LIN {X -121.916,Y -35.3508,Z 150,A -165.0667,B 18.8918,C -0.543,E1 18.7459,E2 253.236} C_DIS
LIN {X -120.9463,Y -38.5366,Z 150,A -163.6955,B 18.8921,C -0.5341,E1 18.747,E2 251.8815} C_DIS
LIN {X -119.9614,Y -41.501,Z 150,A -162.2249,B 18.8921,C -0.5321,E1 18.7483,E2 250.4058} C_DIS
LIN {X -118.8466,Y -44.5932,Z 150,A -160.7318,B 18.8922,C -0.5282,E1 18.7498,E2 248.9133} C_DIS
LIN {X -117.5798,Y -47.8353,Z 150,A -158.9657,B 18.8922,C -0.5304,E1 18.7516,E2 247.1268} C_DIS
LIN {X -116.0485,Y -51.4389,Z 150,A -157.3535,B 18.8924,C -0.5202,E1 18.7534,E2 245.5343} C_DIS
LIN {X -114.7529,Y -54.2683,Z 150,A -155.8591,B 18.8924,C -0.5194,E1 18.7552,E2 244.0312} C_DIS
LIN {X -113.2457,Y -57.3455,Z 150,A -154.3749,B 18.8926,C -0.5131,E1 18.757,E2 242.5558} C_DIS
LIN {X -111.799,Y -60.1208,Z 150,A -153.031,B 18.8928,C -0.5069,E1 18.7587,E2 241.2213} C_DIS
LIN {X -110.4443,Y -62.5757,Z 150,A -151.6788,B 18.8928,C -0.5066,E1 18.7606,E2 239.8605} C_DIS
LIN {X -108.6919,Y -65.5715,Z 150,A -150.1817,B 18.893,C -0.5001,E1 18.7627,E2 238.3729} C_DIS
LIN {X -107.0849,Y -68.1648,Z 150,A -148.7203,B 18.893,C -0.4996,E1 18.7649,E2 236.9031} C_DIS
LIN {X -105.5509,Y -70.5162,Z 150,A -147.3842,B 18.893,C -0.4988,E1 18.767,E2 235.5603} C_DIS
LIN {X -103.218,Y -73.889,Z 150,A -145.457,B 18.893,C -0.4969,E1 18.7701,E2 233.6261} C_DIS
LIN {X -100.6383,Y -77.3663,Z 150,A -143.5811,B 18.8932,C -0.4895,E1 18.7732,E2 231.7609} C_DIS
LIN {X -98.1248,Y -80.5302,Z 150,A -141.6075,B 18.8932,C -0.4905,E1 18.7767,E2 229.7716} C_DIS
LIN {X -95.1979,Y -83.9696,Z 150,A -139.6329,B 18.8934,C -0.4838,E1 18.7803,E2 227.8059} C_DIS
LIN {X -92.4686,Y -86.9661,Z 150,A -137.7265,B 18.8934,C -0.4825,E1 18.7839,E2 225.892} C_DIS
LIN {X -89.2114,Y -90.3049,Z 150,A -135.6196,B 18.8935,C -0.4782,E1 18.7881,E2 223.7863} C_DIS
LIN {X -86.3935,Y -93.0038,Z 150,A -133.8465,B 18.8935,C -0.4751,E1 18.7917,E2 222.0129} C_DIS
LIN {X -83.3889,Y -95.707,Z 150,A -132.0307,B 18.8937,C -0.4713,E1 18.7955,E2 220.1992} C_DIS
LIN {X -80.0505,Y -98.5169,Z 150,A -130.1068,B 18.8937,C -0.466,E1 18.7996,E2 218.2816} C_DIS
LIN {X -76.8507,Y -101.0326,Z 150,A -128.2638,B 18.8939,C -0.463,E1 18.8037,E2 216.4388} C_DIS
LIN {X -74.1065,Y -103.0624,Z 150,A -126.8271,B 18.894,C -0.4567,E1 18.8069,E2 215.0148} C_DIS
LIN {X -71.5613,Y -104.8457,Z 150,A -125.3558,B 18.894,C -0.4568,E1 18.8103,E2 213.5362} C_DIS
LIN {X -69.2262,Y -106.4015,Z 150,A -124.0392,B 18.894,C -0.4567,E1 18.8134,E2 212.2143} C_DIS
LIN {X -66.3429,Y -108.2226,Z 150,A -122.5553,B 18.8941,C -0.4524,E1 18.8169,E2 210.7373} C_DIS
LIN {X -63.1923,Y -110.0926,Z 150,A -120.7476,B 18.8941,C -0.4556,E1 18.8213,E2 208.9124} C_DIS
LIN {X -59.684,Y -112.0331,Z 150,A -119.0868,B 18.8942,C -0.4478,E1 18.8253,E2 207.2692} C_DIS
LIN {X -56.7991,Y -113.5227,Z 150,A -117.6166,B 18.8942,C -0.4462,E1 18.829,E2 205.7988} C_DIS
LIN {X -53.6526,Y -115.0418,Z 150,A -116.1734,B 18.8944,C -0.4395,E1 18.8326,E2 204.3712} C_DIS
LIN {X -51.1576,Y -116.1743,Z 150,A -114.7795,B 18.8944,C -0.4438,E1 18.8362,E2 202.9594} C_DIS
LIN {X -48.581,Y -117.2735,Z 150,A -113.5155,B 18.8944,C -0.4425,E1 18.8394,E2 201.6956} C_DIS
LIN {X -45.6863,Y -118.4311,Z 150,A -111.9655,B 18.8943,C -0.4464,E1 18.8435,E2 200.1291} C_DIS
LIN {X -41.2919,Y -120.0339,Z 150,A -109.958,B 18.8943,C -0.4407,E1 18.8487,E2 198.1337} C_DIS
LIN {X -38.3364,Y -121.0103,Z 150,A -108.5513,B 18.8944,C -0.4397,E1 18.8525,E2 196.7267} C_DIS
LIN {X -34.7483,Y -122.09,Z 150,A -106.9663,B 18.8945,C -0.4346,E1 18.8567,E2 195.1539} C_DIS
LIN {X -32.0597,Y -122.8239,Z 150,A -105.6409,B 18.8945,C -0.4363,E1 18.8603,E2 193.8206} C_DIS
LIN {X -29.1457,Y -123.5476,Z 150,A -104.2669,B 18.8945,C -0.4363,E1 18.864,E2 192.4443} C_DIS
LIN {X -26.2911,Y -124.1859,Z 150,A -102.8898,B 18.8945,C -0.4377,E1 18.8678,E2 191.0603} C_DIS
LIN {X -22.9458,Y -124.8477,Z 150,A -101.4811,B 18.8945,C -0.4322,E1 18.8716,E2 189.6664} C_DIS
LIN {X -20.1813,Y -125.325,Z 150,A -100.1358,B 18.8945,C -0.4347,E1 18.8754,E2 188.3116} C_DIS
LIN {X -16.805,Y -125.8206,Z 150,A -98.5953,B 18.8945,C -0.4344,E1 18.8796,E2 186.7706} C_DIS
LIN {X -13.6931,Y -126.1969,Z 150,A -97.2592,B 18.8945,C -0.4312,E1 18.8833,E2 185.4432} C_DIS
LIN {X -10.6058,Y -126.4938,Z 150,A -95.7869,B 18.8945,C -0.4338,E1 18.8874,E2 183.9621} C_DIS
LIN {X -7.8097,Y -126.6972,Z 150,A -94.4759,B 18.8945,C -0.4354,E1 18.8911,E2 182.6452} C_DIS
LIN {X -4.7122,Y -126.8504,Z 150,A -93.0336,B 18.8945,C -0.4371,E1 18.8951,E2 181.1973} C_DIS
LIN {X -0.0129,Y -126.9396,Z 150,A -90.8917,B 18.8945,C -0.4382,E1 18.9011,E2 179.0522} C_DIS
LIN {X -0.0129,Y -126.9396,Z 150,A -90.8917,B 18.8945,C -0.4382,E1 18.9011,E2 179.0522} C_DIS
Enddeposition()
LIN {X 0.9445,Y -132.9315,Z 151,A -92.5169,B 24.9675,C -1.3177,E1 25.002,E2 179.035} C_DIS
Startdeposition()
$VEL.CP = VEL_PRINT
LIN {X -1.8671,Y -132.9249,Z 151,A -94.2914,B 24.9689,C -1.2879,E1 24.9969,E2 180.8802} C_DIS
LIN {X -5.6543,Y -132.8181,Z 151,A -95.9525,B 24.969,C -1.2863,E1 24.9922,E2 182.5455} C_DIS
LIN {X -9.6665,Y -132.5856,Z 151,A -97.5937,B 24.9688,C -1.291,E1 24.9877,E2 184.176} C_DIS
LIN {X -13.5665,Y -132.245,Z 151,A -99.3804,B 24.969,C -1.2859,E1 24.9827,E2 185.9756} C_DIS
LIN {X -17.278,Y -131.8098,Z 151,A -100.8978,B 24.9688,C -1.2911,E1 24.9785,E2 187.4819} C_DIS
LIN {X -21.1198,Y -131.2512,Z 151,A -102.6961,B 24.9691,C -1.285,E1 24.9735,E2 189.2961} C_DIS
LIN {X -24.96,Y -130.5731,Z 151,A -104.2521,B 24.9687,C -1.2921,E1 24.9692,E2 190.8369} C_DIS
LIN {X -28.3813,Y -129.8728,Z 151,A -105.8606,B 24.969,C -1.2875,E1 24.9648,E2 192.4583} C_DIS
LIN {X -32.5196,Y -128.8985,Z 151,A -107.6687,B 24.9688,C -1.2898,E1 24.9599,E2 194.2635} C_DIS
LIN {X -36.6057,Y -127.8003,Z 151,A -109.609,B 24.9691,C -1.285,E1 24.9547,E2 196.2182} C_DIS
LIN {X -40.6138,Y -126.5814,Z 151,A -111.2002,B 24.9685,C -1.2973,E1 24.9505,E2 197.7829} C_DIS
LIN {X -43.857,Y -125.4948,Z 151,A -112.6685,B 24.9685,C -1.2989,E1 24.9466,E2 199.2504} C_DIS
LIN {X -46.788,Y -124.4315,Z 151,A -114.0517,B 24.9685,C -1.2981,E1 24.943,E2 200.6381} C_DIS
LIN {X -50.015,Y -123.1701,Z 151,A -115.5499,B 24.9684,C -1.2994,E1 24.9391,E2 202.1366} C_DIS
LIN {X -53.1485,Y -121.8511,Z 151,A -116.9929,B 24.9682,C -1.3021,E1 24.9354,E2 203.5766} C_DIS
LIN {X -56.0796,Y -120.5298,Z 151,A -118.3794,B 24.9682,C -1.3037,E1 24.9319,E2 204.9628} C_DIS
LIN {X -59.0775,Y -119.089,Z 151,A -119.8568,B 24.9682,C -1.3032,E1 24.9281,E2 206.445} C_DIS
LIN {X -62.3798,Y -117.3943,Z 151,A -121.5943,B 24.9684,C -1.2984,E1 24.9238,E2 208.1988} C_DIS
LIN {X -66.2634,Y -115.2479,Z 151,A -123.4924,B 24.9683,C -1.3018,E1 24.9192,E2 210.0942} C_DIS
LIN {X -70.015,Y -113.0077,Z 151,A -125.3308,B 24.968,C -1.307,E1 24.9148,E2 211.9262} C_DIS
LIN {X -73.5554,Y -110.736,Z 151,A -127.1913,B 24.968,C -1.3075,E1 24.9105,E2 213.7914} C_DIS
LIN {X -77.2792,Y -108.1697,Z 151,A -129.1146,B 24.9678,C -1.3121,E1 24.9061,E2 215.7103} C_DIS
LIN {X -80.9626,Y -105.4414,Z 151,A -131.1086,B 24.9676,C -1.3148,E1 24.9016,E2 217.7051} C_DIS
LIN {X -84.3353,Y -102.7637,Z 151,A -132.9238,B 24.9673,C -1.3203,E1 24.8977,E2 219.514} C_DIS
LIN {X -87.6541,Y -99.9482,Z 151,A -134.8177,B 24.9673,C -1.3232,E1 24.8937,E2 221.4086} C_DIS
LIN {X -90.8751,Y -97.0289,Z 151,A -136.7418,B 24.9671,C -1.3246,E1 24.8897,E2 223.3371} C_DIS
LIN {X -94.1391,Y -93.8649,Z 151,A -138.6181,B 24.9667,C -1.3329,E1 24.886,E2 225.2015} C_DIS
LIN {X -96.4005,Y -91.5417,Z 151,A -140.0924,B 24.9667,C -1.3322,E1 24.8832,E2 226.6838} C_DIS
LIN {X -99.3357,Y -88.3478,Z 151,A -142.0182,B 24.9667,C -1.3337,E1 24.8795,E2 228.6145} C_DIS
LIN {X -102.2616,Y -84.9433,Z 151,A -143.9468,B 24.9664,C -1.3386,E1 24.8761,E2 230.5403} C_DIS
LIN {X -105.1814,Y -81.2999,Z 151,A -145.9667,B 24.9662,C -1.3432,E1 24.8726,E2 232.5588} C_DIS
LIN {X -107.5667,Y -78.1164,Z 151,A -147.6849,B 24.966,C -1.3474,E1 24.8697,E2 234.2755} C_DIS
LIN {X -110.2226,Y -74.3222,Z 151,A -149.6803,B 24.9657,C -1.3526,E1 24.8666,E2 236.2683} C_DIS
LIN {X -112.5862,Y -70.691,Z 151,A -151.5143,B 24.9654,C -1.3592,E1 24.8638,E2 238.0958} C_DIS
LIN {X -114.6926,Y -67.2189,Z 151,A -153.2996,B 24.9652,C -1.3622,E1 24.8613,E2 239.883} C_DIS
LIN {X -116.8545,Y -63.3868,Z 151,A -155.2497,B 24.9652,C -1.3649,E1 24.8586,E2 241.837} C_DIS
LIN {X -118.5673,Y -60.1173,Z 151,A -156.7268,B 24.9646,C -1.375,E1 24.8568,E2 243.2981} C_DIS
LIN {X -120.0809,Y -57.0343,Z 151,A -158.2751,B 24.9646,C -1.3759,E1 24.8549,E2 244.8525} C_DIS
LIN {X -122.074,Y -52.6328,Z 151,A -160.1615,B 24.9637,C -1.3915,E1 24.8528,E2 246.7121} C_DIS
LIN {X -124.6527,Y -46.1973,Z 151,A -163.3074,B 24.9637,C -1.3928,E1 24.8495,E2 249.8726} C_DIS
LIN {X -125.6967,Y -43.2747,Z 151,A -164.6323,B 24.9634,C -1.3974,E1 24.8483,E2 251.1939} C_DIS
LIN {X -126.6555,Y -40.3817,Z 151,A -165.9957,B 24.9634,C -1.3991,E1 24.8471,E2 252.5612} C_DIS
LIN {X -127.6524,Y -37.1109,Z 151,A -167.4521,B 24.963,C -1.4045,E1 24.8459,E2 254.0131} C_DIS
LIN {X -128.4934,Y -34.0849,Z 151,A -168.8,B 24.9628,C -1.409,E1 24.845,E2 255.3581} C_DIS
LIN {X -129.2828,Y -30.9567,Z 151,A -170.2184,B 24.9627,C -1.412,E1 24.844,E2 256.7776} C_DIS
LIN {X -129.9898,Y -27.8391,Z 151,A -171.6447,B 24.9625,C -1.4141,E1 24.8431,E2 258.2074} C_DIS
LIN {X -130.7638,Y -23.9462,Z 151,A -173.497,B 24.9626,C -1.4128,E1 24.8422,E2 260.0739} C_DIS
LIN {X -131.4438,Y -19.8769,Z 151,A -175.2146,B 24.9622,C -1.4214,E1 24.8414,E2 261.7811} C_DIS
LIN {X -132.0007,Y -15.7532,Z 151,A -177.5065,B 24.9631,C -1.4035,E1 24.8406,E2 264.1294} C_DIS
LIN {X -132.4664,Y -11.1815,Z 151,A -178.8932,B 24.9612,C -1.4383,E1 24.8403,E2 265.4415} C_DIS
LIN {X -132.6968,Y -7.998,Z 151,A 179.6804,B 24.9612,C -1.4403,E1 24.84,E2 266.8716} C_DIS
LIN {X -132.8791,Y -3.952,Z 151,A 177.8291,B 24.9612,C -1.441,E1 24.8398,E2 268.7323} C_DIS
LIN {X -132.9394,Y 0.3425,Z 151,A 175.8798,B 24.961,C -1.4424,E1 24.8398,E2 270.6901} C_DIS
LIN {X -132.8768,Y 4.0338,Z 151,A 174.3565,B 24.9606,C -1.4509,E1 24.8399,E2 272.2023} C_DIS
LIN {X -132.6842,Y 8.2035,Z 151,A 172.6561,B 24.96,C -1.4616,E1 24.8402,E2 273.8875} C_DIS
LIN {X -132.4482,Y 11.3973,Z 151,A 171.2357,B 24.9598,C -1.4643,E1 24.8405,E2 275.3101} C_DIS
LIN {X -132.0267,Y 15.5357,Z 151,A 169.4386,B 24.9595,C -1.47,E1 24.841,E2 277.1043} C_DIS
LIN {X -131.5825,Y 18.9314,Z 151,A 167.9378,B 24.9593,C -1.4737,E1 24.8416,E2 278.6053} C_DIS
LIN {X -130.9707,Y 22.7908,Z 151,A 166.1382,B 24.9593,C -1.4737,E1 24.8424,E2 280.4155} C_DIS
LIN {X -130.2379,Y 26.6541,Z 151,A 164.5648,B 24.9587,C -1.485,E1 24.8432,E2 281.9712} C_DIS
LIN {X -129.5355,Y 29.8826,Z 151,A 163.1173,B 24.9585,C -1.4886,E1 24.8441,E2 283.4187} C_DIS
LIN {X -128.5334,Y 33.935,Z 151,A 161.2667,B 24.9583,C -1.492,E1 24.8454,E2 285.2721} C_DIS
LIN {X -127.581,Y 37.355,Z 151,A 159.7557,B 24.958,C -1.4978,E1 24.8466,E2 286.7778} C_DIS
LIN {X -126.591,Y 40.5836,Z 151,A 158.3104,B 24.9577,C -1.503,E1 24.8478,E2 288.2192} C_DIS
LIN {X -125.5355,Y 43.7396,Z 151,A 156.8746,B 24.9574,C -1.5075,E1 24.8491,E2 289.6524} C_DIS
LIN {X -124.3586,Y 46.9825,Z 151,A 155.3885,B 24.9572,C -1.5122,E1 24.8505,E2 291.1356} C_DIS
LIN {X -123.1961,Y 49.9507,Z 151,A 153.9376,B 24.9572,C -1.5129,E1 24.852,E2 292.5931} C_DIS
LIN {X -121.4213,Y 54.1216,Z 151,A 151.3837,B 24.9584,C -1.4904,E1 24.855,E2 295.2147} C_DIS
LIN {X -119.3267,Y 58.5956,Z 151,A 149.7576,B 24.9567,C -1.5208,E1 24.8569,E2 296.7771} C_DIS
LIN {X -117.2338,Y 62.6823,Z 151,A 147.7912,B 24.9563,C -1.5273,E1 24.8594,E2 298.7384} C_DIS
LIN {X -115.1797,Y 66.3812,Z 151,A 145.969,B 24.956,C -1.5328,E1 24.8619,E2 300.557} C_DIS
LIN {X -113.0168,Y 70.0003,Z 151,A 144.1151,B 24.9558,C -1.5364,E1 24.8646,E2 302.412} C_DIS
LIN {X -110.6952,Y 73.6166,Z 151,A 142.2441,B 24.9555,C -1.5408,E1 24.8674,E2 304.2819} C_DIS
LIN {X -108.2732,Y 77.1345,Z 151,A 140.3914,B 24.9553,C -1.5454,E1 24.8704,E2 306.1327} C_DIS
LIN {X -105.7719,Y 80.5305,Z 151,A 138.5956,B 24.9549,C -1.5515,E1 24.8734,E2 307.9227} C_DIS
LIN {X -103.137,Y 83.8786,Z 151,A 136.7421,B 24.9547,C -1.5556,E1 24.8766,E2 309.775} C_DIS
Enddeposition()
END
